(* CODESYS project tc3_hbi_system.library
   Company: BeckHoff
   DefaultNamespace: Tc3_HBI_System
   Version: 3.3.2.1
   Placeholder: Tc3_HBI_System
   Title: Tc3_HBI_System

Project tree, tasks and I/O mapping:
  libraries: Tc2_EtherCAT, * (Beckhoff Automation GmbH); Tc2_IoFunctions, * (Beckhoff Automation GmbH); Tc2_Standard, * (Beckhoff Automation GmbH); Tc2_SUPS, * (Beckhoff Automation GmbH); Tc2_System, * (Beckhoff Automation GmbH); Tc2_Utilities, * (Beckhoff Automation GmbH); Tc3_Interfaces, * (Beckhoff Automation GmbH); Tc3_Module, * (Beckhoff Automation GmbH)
  DUTs/
  GVLs/
  POUs/
    BASIC/
      POUs/
        FBs/
          DUTs/
            data type ST_Basic
            data type ST_Basic_Status
          GVLs/
            global variables GVL_Basic
          ITFs/
            interface I_Basic: M_nError, M_nReset, P_bAuto, P_bError, P_bManual, P_bReady, P_bReset, P_nErrorID
          function block FB_Basic [ST]: M_nError, M_nReset, P_bAuto, P_bError, P_bManual, P_bReady, P_bReset, P_nErrorID
    FileSystem/
      ITFs/
        interface I_FileSystem: P_sDirectoryPath, P_sSubDirPath
      DUTs/
        data type ST_FileSystem
      function block FB_FileAccess [ST]: M_nDirectory, M_nSequence, M_sGetToken, P_sDirectoryPath, P_sSubDirPath
    SYSTEM/
      POUs/
        FBs/
          EtherCAT/
            DUTs/
              HW/
                data type ST_EtherCAT_HW_IN
                data type ST_EtherCAT_HW_TerminalDiagInfo
              data type ST_EtherCAT_Diag
              data type ST_EtherCAT_HW_Diag
            GVLs/
              global variables GVL_EtherCAT_Diag
            ITFs/
              interface I_EtherCAT_Diag: M_nCyclic, P_bEtherCAT_Ok, P_bWcError, P_nCfgSlaveCount, P_nDevState, P_nSlaveCounts
            function block FB_EtherCAT_Diag [ST]: M_nCyclic, M_sGetToken, P_bEtherCAT_Ok, P_bWcError, P_nCfgSlaveCount, P_nDevState, P_nSlaveCounts
          NovRam/
            DUTs/
              data type ST_NovRam
            ITFs/
              interface I_NovRam: M_nEnable
            function block FB_NovRam [ST]: M_nEnable, M_nRead, M_nWrite
          Persistent/
            DUTs/
              data type ST_WritePersistentData
            ITFs/
              interface I_WritePersistentData: M_n1_Second_UPS, M_nEnable, M_nWrite, P_bBusy, P_bPowerFailDetect, P_eSUPS_Mode, P_nWriteCNT
            function block FB_WritePersistentData [ST]: M_n1_Second_UPS, M_nEnable, M_nWrite, P_bBusy, P_bPowerFailDetect, P_eSUPS_Mode, P_nWriteCNT
          System/
            DUTs/
              data type ST_System
            ITFs/
              interface I_System: M_nCerHost, M_nEnable, M_nGetTimeStampInMs, P_bIs_ARM, P_bIs_CE_Device, P_bIs_x64, P_bIs_x86, P_nAdsPort, P_nCycleTime, P_stDeviceIdentificationEx, P_sTwinCAT_Version
            function block FB_System [ST]: M_nCerHost, M_nEnable, M_nGetTimeStampInMs, P_bIs_ARM, P_bIs_CE_Device, P_bIs_x64, P_bIs_x86, P_nAdsPort, P_nCycleTime, P_stDeviceIdentificationEx, P_sTwinCAT_Version
  Version/
    global variables Global_Version
  VISUs/
  Tc3_HBI_System.tmc
*)

// POUs/BASIC/POUs/FBs/DUTs/ST_Basic
TYPE ST_Basic :
STRUCT
	bAuto: BOOL;
	bManual: BOOL;
	bReady: BOOL;
	bReset: BOOL;
	bError: BOOL;
	nErrorID: UDINT;
	nStatus: UDINT;	
	arr_nStatus: ARRAY[1..20] OF UDINT;
END_STRUCT
END_TYPE

// POUs/BASIC/POUs/FBs/DUTs/ST_Basic_Status
TYPE ST_Basic_Status :
STRUCT
	nError: UDINT;
	nReset:UDINT;
END_STRUCT
END_TYPE

// POUs/FileSystem/DUTs/ST_FileSystem
TYPE ST_FileSystem :
STRUCT
END_STRUCT
END_TYPE

// POUs/SYSTEM/POUs/FBs/EtherCAT/DUTs/HW/ST_EtherCAT_HW_IN
TYPE ST_EtherCAT_HW_IN :
STRUCT
	AI_AmsNetId: AMSNETID;
	AI_nDevState: UINT;
	AI_nCfgSlaveCount: UINT;							
	AI_nSlaveCounts: UINT;								
	AI_nFrmXWcState: ARRAY[0..(GVL_EtherCAT_Diag.MAX_NUMBERS_OF_EC_FRAMES -1)] OF UINT;
END_STRUCT
END_TYPE

// POUs/SYSTEM/POUs/FBs/EtherCAT/DUTs/HW/ST_EtherCAT_HW_TerminalDiagInfo
TYPE ST_EtherCAT_HW_TerminalDiagInfo :
STRUCT
	nAddr: UINT;
	sType: STRING(50);
	sName: STRING(50);
	nDeviceState: BYTE;
	nLinkState: BYTE;
END_STRUCT
END_TYPE

// POUs/SYSTEM/POUs/FBs/EtherCAT/DUTs/ST_EtherCAT_Diag
TYPE ST_EtherCAT_Diag EXTENDS ST_Basic:
STRUCT
	bEtherCAT_Ok: BOOL;				// ErtherCAT Ok signal
	bWcError: BOOL;
	nDevState: UINT;
	nCfgSlaveCount: UINT;							
	nSlaveCounts: UINT;								
END_STRUCT
END_TYPE

// POUs/SYSTEM/POUs/FBs/EtherCAT/DUTs/ST_EtherCAT_HW_Diag
TYPE ST_EtherCAT_HW_Diag :
STRUCT
	stAmsNetId: AMSNETID;			// EtherCAT Ams net id
	nState: WORD;					// EtherCAT master state
	sState: STRING;					// EtherCAT master state (string)
	nDevState: UINT;				// EtherCAT master DevState
	sDevState: STRING;				// EtherCAT master DevState (string)
	nCfgSlaveCount: UINT;			// Project configured slaves
	nSlaveCounts: UINT;				// Actual slave counts
	nMaxNumberOfSlaves: UINT;		// Max numbers of EtherCAT slaves
	bWcError: BOOL;					// Wc error
	bEtherCAT_Ok: BOOL;				// ErtherCAT Ok signal
	bReady: BOOL;					// Ready
	bError: BOOL;					// Error
	nErrorID: UDINT;				// Error ID
	arrFrmXWcState: ARRAY[0..(GVL_EtherCAT_Diag.MAX_NUMBERS_OF_EC_FRAMES - 1)] OF UINT;		// EtherCAT master Wc state
	arrEcTerminalDiagInfo: ARRAY[1..GVL_EtherCAT_Diag.MAX_NUMBERS_OF_EC_SLAVES] OF ST_EtherCAT_HW_TerminalDiagInfo;
END_STRUCT
END_TYPE

// POUs/SYSTEM/POUs/FBs/NovRam/DUTs/ST_NovRam
TYPE ST_NovRam EXTENDS ST_Basic :
STRUCT
	bEnable: BOOL;
END_STRUCT
END_TYPE

// POUs/SYSTEM/POUs/FBs/Persistent/DUTs/ST_WritePersistentData
TYPE ST_WritePersistentData EXTENDS ST_Basic :
STRUCT
	bWrite: BOOL;
	bBusy: BOOL;
	bPowerFailDetect: BOOL;
	nWriteCNT: UDINT;
END_STRUCT
END_TYPE

// POUs/SYSTEM/POUs/FBs/System/DUTs/ST_System
TYPE ST_System EXTENDS ST_Basic :
STRUCT
	bIs_CE_Device: BOOL;			// Is a CE Device
	bIs_ARM: BOOL;					// Is ARM runtime
	bIs_x86: BOOL;					// Is x86 runtime
	bIs_x64: BOOL;					// Is x64 runtime
	nAdsPort: UINT;					// Plc port nr
	nCycleTime: UDINT;				// Plc cycle time in 100nS
	bCerHost_Enable: BOOL;			// Enable CerHost
	bCerHost_Disable: BOOL;			// Disable CerHost
	sTwinCAT_Version: STRING(20);	// Runtime version
	stDeviceIdentificationEx: Tc2_Utilities.ST_DeviceIdentificationEx;
END_STRUCT
END_TYPE

// POUs/BASIC/POUs/FBs/GVLs/GVL_Basic
VAR_GLOBAL CONSTANT
	cIDLE: UDINT:= 0;						//	0 = idle
	cCOUPLED: UDINT:= 1;					//	1 = coupled
	cSTARTING: UDINT:= 2;					//	2 = starting
	cRUNNING: UDINT:= 3;					//	3 = running
	cABORTED: UDINT:= 4;					//	4 = aborted
	cNO_HARDWARE_CONNECTED: UDINT:= 5;		// 	5 = no hardware connected

	cPOINTER_OR_INDEX_ERROR: UDINT:= 7;		//	7 = pointer or index error
	cMAPPING_ERROR: UDINT:= 8;				//	8 = mapping error
	cPARAMETER_ERROR: UDINT:= 9;			//	9 = parameter error
	cCOMPLETE: UDINT:= 10;					//	10 = complete
END_VAR

// POUs/SYSTEM/POUs/FBs/EtherCAT/GVLs/GVL_EtherCAT_Diag
{attribute 'qualified_only'}
VAR_GLOBAL CONSTANT
	MAX_NUMBERS_OF_EC_SLAVES: UINT:= 1000;		// Max numbers of EtherCAT slaves
	MAX_NUMBERS_OF_EC_FRAMES: UINT:= 10;		// Max numbers of EtherCAT frames
END_VAR

// Version/Global_Version
{attribute 'TcGenerated'}
// This function has been automatically generated from the project information.
VAR_GLOBAL CONSTANT
	{attribute 'const_non_replaced'}
	{attribute 'linkalways'}
	stLibVersion_Tc3_HBI_System : ST_LibVersion := (iMajor := 3, iMinor := 3, iBuild := 2, iRevision := 1, sVersion := '3.3.2.1');
END_VAR

// POUs/BASIC/POUs/FBs/ITFs/I_Basic
INTERFACE I_Basic

//	The result of the method is an unsigned double integer
//	0 = idle 
//	1 = coupled
//	2 = starting
//	3 = running
//	4 = aborted
// 	5 = no hardware connected
//  6 = Spare
//	7 = pointer or index error
//	8 = mapping error
//	9 = parameter error
//	10 = complete
//	Any other number = ErrorID
METHOD PUBLIC M_nError : UDINT
VAR_INPUT
	nErrorID: UDINT;
END_VAR
END_METHOD

//	The result of the method is an unsigned double integer
//	0 = idle 
//	1 = coupled
//	2 = starting
//	3 = running
//	4 = aborted
// 	5 = no hardware connected
//  6 = Spare
//	7 = pointer or index error
//	8 = mapping error
//	9 = parameter error
//	10 = complete
//	Any other number = ErrorID
METHOD PUBLIC M_nReset : UDINT
VAR_INPUT
	bExecute: BOOL;
END_VAR
END_METHOD

PROPERTY PUBLIC P_bAuto : BOOL
GET
END_GET
SET
END_SET
END_PROPERTY

PROPERTY PUBLIC P_bError : BOOL
GET
END_GET
END_PROPERTY

PROPERTY PUBLIC P_bManual : BOOL
GET
END_GET
SET
END_SET
END_PROPERTY

PROPERTY PUBLIC P_bReady : BOOL
GET
END_GET
SET
END_SET
END_PROPERTY

PROPERTY PUBLIC P_bReset : BOOL
GET
END_GET
END_PROPERTY

PROPERTY PUBLIC P_nErrorID : UDINT
GET
END_GET
END_PROPERTY

END_INTERFACE

// POUs/BASIC/POUs/FBs/FB_Basic
//------------------------------------------------------------------------------------------
//                                                                                        	
//***************************** Beckhoff TwinCAT Examples **********************************
//                                                                                        	
//************************************* WARNING ********************************************
// This program is only an example. If it is used as a control program in any real        	
// application, Beckhoff is not responsible for any malfunction, loss or damage           	
// which could arise by using this program!                                               	
//                                                                                        	
//*************************************  Program Info. *************************************
//                                                                                        	
// PLC program name:       	FB_Basic (FB)               	                           	
// Hardware platform:      	TwinCat v3.1.4022				                          	                                  	
//                                                                                        	
// ======================================================================================== 
//         Version       Date                        Remarks                              	
// ======================================================================================== 
//         3.1           27 feb 2018                 First release of this example        	    	
// ======================================================================================== 
//                                                                                        	
//******************************* Aims OF this PLC PROGRAM *********************************
//                                                                                        	
// Basic FB  						 			                               	
//																	                      	
//                                                                                        	
//----------------------------------------------------------------------------------------- 
FUNCTION_BLOCK FB_Basic IMPLEMENTS I_Basic
VAR
	_iIdx: INT;		// Temporary variabel - Index pointer
	
//*************************
// Property variables
//*************************
	_bReset: BOOL;
	_bAuto: BOOL := TRUE;
	_bManual: BOOL;
	_bError: BOOL;
	_nErrorID: UDINT;
	_bReady: BOOL;
	
//*************************
// Methods variable
//*************************
	FB_Basic_M_nReset_nScanCNT: UINT;
	FB_Basic_M_nReset_fbR_TRIG: Tc2_Standard.R_TRIG;
END_VAR

//	The result of the method is an unsigned double integer
//	0 = idle 
//	1 = coupled
//	2 = starting
//	3 = running
//	4 = aborted
// 	5 = no hardware connected
//  6 = Spare
//	7 = pointer or index error
//	8 = mapping error
//	9 = parameter error
//	10 = complete
//	Any other number = ErrorID
METHOD PUBLIC M_nError : UDINT
VAR_INPUT
	nErrorID: UDINT;
END_VAR
//**********************************
// Update error
//**********************************
IF NOT _bReset THEN
	IF NOT _bError THEN
		_nErrorID:= nErrorID;
		_bError:= TRUE;
	END_IF
END_IF

M_nError:= cCOMPLETE;
END_METHOD

//	The result of the method is an unsigned double integer
//	0 = idle 
//	1 = coupled
//	2 = starting
//	3 = running
//	4 = aborted
// 	5 = no hardware connected
//  6 = Spare
//	7 = pointer or index error
//	8 = mapping error
//	9 = parameter error
//	10 = complete
//	Any other number = ErrorID
METHOD PUBLIC M_nReset : UDINT
VAR_INPUT
	bExecute: BOOL;
END_VAR
//**********************************
// Wait for execute
//**********************************
FB_Basic_M_nReset_fbR_TRIG(CLK:= bExecute);
IF FB_Basic_M_nReset_fbR_TRIG.Q THEN
	FB_Basic_M_nReset_nScanCNT:= 4;	
	_bReset:= TRUE;
ELSE
	// Delay
	IF FB_Basic_M_nReset_nScanCNT = 0 THEN
		IF NOT bExecute THEN
			_bReset:= FALSE;
		END_IF
	ELSE
		IF FB_Basic_M_nReset_nScanCNT <= 2 THEN
			_bError:= FALSE;
			_nErrorID:= 16#00;
		END_IF	
	END_IF

	// Scan counter
	IF FB_Basic_M_nReset_nScanCNT > 0 THEN
		FB_Basic_M_nReset_nScanCNT:= FB_Basic_M_nReset_nScanCNT -1;
	ELSE	
		FB_Basic_M_nReset_nScanCNT:= 0;
	END_IF

	// Return method state
	IF bExecute THEN
		IF FB_Basic_M_nReset_nScanCNT = 0 THEN
			M_nReset:= cCOMPLETE;
		ELSE
			M_nReset:= cRUNNING;
		END_IF
	ELSE	
		M_nReset:= cIDLE;
	END_IF	
END_IF
END_METHOD

PROPERTY PUBLIC P_bAuto : BOOL
GET
P_bAuto:= _bAuto;
END_GET
SET
_bAuto:= P_bAuto;
END_SET
END_PROPERTY

PROPERTY PUBLIC P_bError : BOOL
GET
P_bError:= _bError;
END_GET
END_PROPERTY

PROPERTY PUBLIC P_bManual : BOOL
GET
P_bManual:= _bManual;
END_GET
SET
_bManual:= P_bManual;
END_SET
END_PROPERTY

PROPERTY PUBLIC P_bReady : BOOL
GET
P_bReady:= _bReady;
END_GET
SET
PUBLIC 
VAR
END_VAR
_bReady:= P_bReady;
END_SET
END_PROPERTY

PROPERTY PUBLIC P_bReset : BOOL
GET
P_bReset:= _bReset;
END_GET
END_PROPERTY

PROPERTY PUBLIC P_nErrorID : UDINT
GET
P_nErrorID:= _nErrorID;
END_GET
END_PROPERTY

END_FUNCTION_BLOCK

// POUs/FileSystem/ITFs/I_FileSystem
INTERFACE I_FileSystem EXTENDS I_Basic

PROPERTY P_sDirectoryPath : T_MaxString
GET
END_GET
SET
END_SET
END_PROPERTY

PROPERTY P_sSubDirPath : T_MaxString
GET
END_GET
SET
END_SET
END_PROPERTY

END_INTERFACE

// POUs/FileSystem/FB_FileAccess
FUNCTION_BLOCK PUBLIC FB_FileAccess EXTENDS FB_Basic IMPLEMENTS I_FileSystem
VAR_INPUT
END_VAR
VAR_OUTPUT
END_VAR
VAR
	// Directory
	FB_FileAccess_DirectoryPath:	T_MAXSTRING:='C:\';
	FB_FileAccess_SubDirPath:		T_MAXSTRING:='AEM\Data\ControllerLog';
	fbCreateDir			: FB_CreateDir;
	fbEnumFindFileEntry	: FB_EnumFindFileEntry;
	
	FB_FileAccess_M_nDirectory_iState	: INT;
	FB_FileAccess_M_nDirectory_bExecute: BOOL;
	FB_FileAccess_M_nDirectory_fbExecute: R_TRIG;
	
	FB_FileAccess_M_nSequence_iState	: INT;
	FB_FileAccess_M_nSequence_bExecute: BOOL;
	FB_FileAccess_M_nSequence_fbExecute: R_TRIG;
	FB_FileAccess_M_nSequence_sPathName:	T_MAXSTRING:='C:\AEM\Data\ControllerLog';
	
	FB_FileAccess_M_nDirectory_sSubDirPath: T_MAXSTRING;
	FB_FileAccess_M_nDirectory_sSubDirPath1: T_MAXSTRING;
	FB_FileAccess_M_nDirectory_sSubDirPath2: T_MAXSTRING;
	FB_FileAccess_M_nDirectory_sSubDirPath3: T_MAXSTRING;
	FB_FileAccess_M_nDirectory_sSubDirPath4: T_MAXSTRING;
	FB_FileAccess_M_nDirectory_nToken	   : INT;	
END_VAR

METHOD PUBLIC M_nDirectory : UDINT
VAR_INPUT
	bExecute: BOOL;
END_VAR
VAR	
END_VAR
FB_FileAccess_M_nDirectory_bExecute:= bExecute;
FB_FileAccess_M_nDirectory_fbExecute(CLK:= FB_FileAccess_M_nDirectory_bExecute, Q=> );

IF FB_FileAccess_M_nDirectory_fbExecute.Q THEN
	FB_FileAccess_M_nDirectory_iState:= 10;
END_IF

	FB_FileAccess_M_nDirectory_sSubDirPath1:= M_sGetToken(sAllTokens:= FB_FileAccess_SubDirPath, nToken:= 1, sDelim:= '\');
	FB_FileAccess_M_nDirectory_sSubDirPath2:= M_sGetToken(sAllTokens:= FB_FileAccess_SubDirPath, nToken:= 2, sDelim:= '\');
	FB_FileAccess_M_nDirectory_sSubDirPath3:= M_sGetToken(sAllTokens:= FB_FileAccess_SubDirPath, nToken:= 3, sDelim:= '\');
	FB_FileAccess_M_nDirectory_sSubDirPath4:= M_sGetToken(sAllTokens:= FB_FileAccess_SubDirPath, nToken:= 4, sDelim:= '\');
	
	IF FB_FileAccess_M_nDirectory_sSubDirPath1='' OR FB_FileAccess_M_nDirectory_sSubDirPath2= '' OR FB_FileAccess_M_nDirectory_sSubDirPath3=''
			OR FB_FileAccess_M_nDirectory_sSubDirPath4<> '' THEN
		M_nError(nErrorID:= cPARAMETER_ERROR);
		M_nDirectory:= cPARAMETER_ERROR;
		RETURN;
	END_IF
	
IF _bReset THEN
	IF _bError THEN
		FB_FileAccess_M_nDirectory_iState:= 0;
	END_IF
END_IF

CASE FB_FileAccess_M_nDirectory_iState OF
 
	0: // Init
		M_nDirectory:= cIDLE;
		
		M_nSequence(bExecute:= FALSE, sPathName:= 'C:\AEM\Data\ControllerLog');
		FB_FileAccess_M_nDirectory_iState:= 1;
		
	1: // Waiting for execute
		;
		
	10: // Create directory
	
		M_nDirectory:= cRUNNING;
		
		IF M_nSequence(bExecute:= TRUE, sPathName:= CONCAT(FB_FileAccess_DirectoryPath,FB_FileAccess_M_nDirectory_sSubDirPath1))= cComplete THEN
			M_nSequence(bExecute:= FALSE, sPathName:= CONCAT(FB_FileAccess_DirectoryPath,FB_FileAccess_M_nDirectory_sSubDirPath1));
			FB_FileAccess_M_nDirectory_iState:= 20;
			ELSIF _bError THEN
				M_nDirectory:= M_nError(nErrorID:= _nErrorID);
				FB_FileAccess_M_nDirectory_iState:= 999;
		END_IF
	
	20: // Create directory
		M_nDirectory:= cRUNNING;
		IF M_nSequence(bExecute:= TRUE, sPathName:= CONCAT(FB_FileAccess_DirectoryPath,
				CONCAT(FB_FileAccess_M_nDirectory_sSubDirPath1,CONCAT('\',FB_FileAccess_M_nDirectory_sSubDirPath2))))= cComplete THEN
			M_nSequence(bExecute:= FALSE, sPathName:= CONCAT(FB_FileAccess_DirectoryPath,FB_FileAccess_M_nDirectory_sSubDirPath1));
			FB_FileAccess_M_nDirectory_iState:= 30;
			ELSIF _bError THEN
				M_nDirectory:= M_nError(nErrorID:= _nErrorID);
				FB_FileAccess_M_nDirectory_iState:= 999;
		END_IF
	
	30: // Create directory
		M_nDirectory:= cRUNNING;
		IF M_nSequence(bExecute:= TRUE, sPathName:= CONCAT(FB_FileAccess_DirectoryPath,CONCAT(FB_FileAccess_M_nDirectory_sSubDirPath1,
							CONCAT('\',CONCAT(FB_FileAccess_M_nDirectory_sSubDirPath2,CONCAT('\',FB_FileAccess_M_nDirectory_sSubDirPath3))))))= cComplete THEN
			M_nSequence(bExecute:= FALSE, sPathName:= CONCAT(FB_FileAccess_DirectoryPath,FB_FileAccess_M_nDirectory_sSubDirPath1));
			FB_FileAccess_M_nDirectory_iState:= 40;
			ELSIF _bError THEN
				M_nDirectory:= M_nError(nErrorID:= _nErrorID);
				FB_FileAccess_M_nDirectory_iState:= 999;
		END_IF
		
	40:
		M_nDirectory:= cComplete;
		
		IF NOT FB_FileAccess_M_nDirectory_bExecute THEN
			FB_FileAccess_M_nDirectory_iState:= 0;
		END_IF
	
	999:// Error state
		M_nSequence(bExecute:= FALSE, sPathName:= CONCAT(FB_FileAccess_DirectoryPath,FB_FileAccess_M_nDirectory_sSubDirPath1));
		
	ELSE FB_FileAccess_M_nDirectory_iState:= 0;
		
END_CASE
END_METHOD

METHOD PUBLIC M_nSequence : UDINT
VAR_INPUT
	bExecute: BOOL;
	sPathName: T_MaxString;
END_VAR
// Local variables
FB_FileAccess_M_nSequence_bExecute:= bExecute;
FB_FileAccess_M_nSequence_sPathName:= sPathName;

IF _bReset THEN
	IF _bError THEN
		FB_FileAccess_M_nSequence_iState:= 0;
	END_IF
END_IF

FB_FileAccess_M_nSequence_fbExecute(CLK:= FB_FileAccess_M_nSequence_bExecute, Q=> );
IF FB_FileAccess_M_nSequence_fbExecute.Q THEN
	FB_FileAccess_M_nSequence_iState:= 10;
END_IF

CASE FB_FileAccess_M_nSequence_iState OF 
	0: // Init
		M_nSequence:= cIDLE;
		
		fbEnumFindFileEntry(sNetId:= '', bExecute:= FALSE, );
		fbCreateDir(sNetId:= '', bExecute:= FALSE, );
		FB_FileAccess_M_nSequence_iState:= 1;
		
	1: // Waiting for execute
		;
		
	10: // Check if directory exit
		M_nSequence:= cRUNNING;
		
		fbEnumFindFileEntry(
			sNetId:= '', 
			sPathName:= FB_FileAccess_M_nSequence_sPathName, 
			eCmd:= eEnumCmd_First, 
			bExecute:= TRUE, 
			tTimeout:= T#5S, 
			bBusy=> , 
			bError=> , 
			nErrID=> , 
			bEOE=> , 
			stFindFile=> );
		IF NOT fbEnumFindFileEntry.bBusy THEN	
			IF fbEnumFindFileEntry.bError THEN
				M_nError(nErrorID:= fbEnumFindFileEntry.nErrId);
				FB_FileAccess_M_nSequence_iState:= 999;
			ELSE
				IF NOT fbEnumFindFileEntry.bEOE THEN
					FB_FileAccess_M_nSequence_iState:= 30; (*target dir is exist*)
					ELSE 
						FB_FileAccess_M_nDirectory_sSubDirPath:= FB_FileAccess_M_nSequence_sPathName;
						FB_FileAccess_M_nSequence_iState:= 20;	(*target dir no exist*)
				END_IF
			END_IF
			fbEnumFindFileEntry(sNetId:= '', bExecute:= FALSE, );
		END_IF	
		
	20: // Create directory
		M_nSequence:= cRUNNING;
		
		fbCreateDir(
			sNetId:= '', 
			sPathName:= FB_FileAccess_M_nSequence_sPathName, 
			ePath:= PATH_GENERIC, 
			bExecute:= TRUE, 
			tTimeout:= T#5S, 
			bBusy=> , 
			bError=> , 
			nErrId=> );
		IF NOT fbCreateDir.bBusy THEN	
			IF fbCreateDir.bError THEN
				M_nError(nErrorID:= fbCreateDir.nErrId);
				FB_FileAccess_M_nSequence_iState:= 999;
			ELSE
				FB_FileAccess_M_nSequence_iState:= 30;	
			END_IF
			fbCreateDir(sNetId:= '', bExecute:= FALSE, );
		END_IF
		
	30: // Complete
		M_nSequence:= cComplete;
		IF NOT FB_FileAccess_M_nSequence_bExecute THEN
			FB_FileAccess_M_nSequence_iState:= 0;
		END_IF
		
	999: // error state
		;
	
	ELSE FB_FileAccess_M_nSequence_iState:= 0;
		
END_CASE
END_METHOD

METHOD PUBLIC M_sGetToken : STRING
VAR_INPUT
	sAllTokens: Tc2_System.T_MaxString;
	nToken: UINT;
  	sDelim: STRING;
END_VAR
VAR
// Temporary Variables 
	pString: POINTER TO STRING;
	nCurTokenLocation: INT;
END_VAR
pString:= ADR(sAllTokens);

IF nToken < 1 OR LEN(sDelim) < 1 THEN
	// Negative OR zeroth token OR empty delimiter strings mean an empty token 
	M_sGetToken:= '';
 	RETURN;
ELSE
	IF nToken = 1 THEN
	// Quickly extract the first token 
	nCurTokenLocation:= FIND(pString^, sDelim);
	   	IF nCurTokenLocation > 1 THEN
	   		M_sGetToken:= LEFT(pString^, nCurTokenLocation - 1);
	   	ELSE
			M_sGetToken:= pString^;
	    END_IF
	ELSE
		// FIND the Nth token 
		REPEAT
			nCurTokenLocation:= FIND(pString^, sDelim);
			IF nCurTokenLocation = 0 THEN
				M_sGetToken:= '';
				RETURN;
			ELSE
				pString:= pString + INT_TO_DWORD(nCurTokenLocation -1) + INT_TO_DWORD(LEN(sDelim));
			END_IF
	
			nToken:= nToken - 1;
			UNTIL nToken = 1
		END_REPEAT;

		// Extract the Nth token (Which is the next token AT this point) 
		nCurTokenLocation:= FIND(pString^, sDelim);
		IF nCurTokenLocation > 0 THEN
			M_sGetToken:= LEFT(pString^, nCurTokenLocation - 1);
			RETURN;
		ELSE
			M_sGetToken:= pString^;
		   	RETURN;
		END_IF
	END_IF
END_IF
END_METHOD

PROPERTY P_sDirectoryPath : T_MaxString
GET
P_sDirectoryPath:= FB_FileAccess_DirectoryPath;
END_GET
SET
FB_FileAccess_DirectoryPath:= P_sDirectoryPath;
END_SET
END_PROPERTY

PROPERTY P_sSubDirPath : T_MaxString
GET
P_sSubDirPath:= FB_FileAccess_SubDirPath;
END_GET
SET
FB_FileAccess_SubDirPath:= P_sSubDirPath;
END_SET
END_PROPERTY

END_FUNCTION_BLOCK

// POUs/SYSTEM/POUs/FBs/EtherCAT/ITFs/I_EtherCAT_Diag
INTERFACE I_EtherCAT_Diag EXTENDS I_Basic

//	The result of the method is an unsigned double integer
//	0 = idle 
//	1 = coupled
//	2 = starting
//	3 = running
//	4 = aborted
// 	5 = no hardware connected
//  6 = Spare
//	7 = pointer or index error
//	8 = mapping error
//	9 = parameter error
//	10 = complete
//	Any other number = ErrorID
METHOD PUBLIC M_nCyclic : UDINT
VAR_INPUT
	bEnable: BOOL;
	pEtherCAT_Diag: POINTER TO ST_EtherCAT_HW_Diag;	
END_VAR
END_METHOD

PROPERTY PUBLIC P_bEtherCAT_Ok : BOOL
GET
END_GET
SET
END_SET
END_PROPERTY

PROPERTY PUBLIC P_bWcError : bool
GET
END_GET
END_PROPERTY

PROPERTY PUBLIC P_nCfgSlaveCount : UINT
GET
END_GET
END_PROPERTY

PROPERTY PUBLIC P_nDevState : UINT
GET
END_GET
END_PROPERTY

PROPERTY PUBLIC P_nSlaveCounts : UINT
GET
END_GET
END_PROPERTY

END_INTERFACE

// POUs/SYSTEM/POUs/FBs/EtherCAT/FB_EtherCAT_Diag
//------------------------------------------------------------------------------------------
//                                                                                        	
//***************************** Beckhoff TwinCAT Examples **********************************
//                                                                                        	
//************************************* WARNING ********************************************
// This program is only an example. If it is used as a control program in any real        	
// application, Beckhoff is not responsible for any malfunction, loss or damage           	
// which could arise by using this program!                                               	
//                                                                                        	
//*************************************  Program Info. *************************************
//                                                                                        	
// PLC program name:       	FB_EtherCAT_Diag (FB)                                          	
// Hardware platform:      	TwinCAT v3.1.4022				                          	                                  	
//                                                                                        	
// ======================================================================================== 
//         Version       Date                        Remarks                              	
// ======================================================================================== 
//         3.1           27 feb 2018                 First release of this example        	
// ======================================================================================== 
//                                                                                        	
//******************************* Aims OF this PLC PROGRAM *********************************
//                                                                                        	
// EtherCAT diagnose				 			                                      	
//																	                      	
//                                                                                        	
//----------------------------------------------------------------------------------------- 
FUNCTION_BLOCK FB_EtherCAT_Diag EXTENDS FB_Basic IMPLEMENTS I_EtherCAT_Diag
VAR
	bFirstScan: BOOL:= TRUE;
	stIN AT %I*: ST_EtherCAT_HW_IN;
	
	_pEtherCAT_Diag: POINTER TO ST_EtherCAT_HW_Diag;	
	_bWcError: BOOL;
	_nDeviceNumber: UINT:= 1;
	
	arrEcSlaveConfigData: ARRAY[1..GVL_EtherCAT_Diag.MAX_NUMBERS_OF_EC_SLAVES] OF Tc2_EtherCAT.ST_EcSlaveConfigData;
	arrEcSlaveState: ARRAY[1..GVL_EtherCAT_Diag.MAX_NUMBERS_OF_EC_SLAVES] OF Tc2_EtherCAT.ST_EcSlaveState;
	arrEcSlaveName: ARRAY[1..GVL_EtherCAT_Diag.MAX_NUMBERS_OF_EC_SLAVES] OF STRING;;

	fbEcGetMasterState: Tc2_EtherCAT.FB_EcGetMasterState;
	fbEcGetConfSlaves: Tc2_EtherCAT.FB_EcGetConfSlaves;
	fbEcGetAllSlaveStates: Tc2_EtherCAT.FB_EcGetAllSlaveStates;
	fbEcGetSlaveIdentity: Tc2_EtherCAT.FB_EcGetSlaveIdentity;
END_VAR

//	The result of the method is an unsigned double integer
//	0 = idle 
//	1 = coupled
//	2 = starting
//	3 = running
//	4 = aborted
// 	5 = no hardware connected
//  6 = Spare
//	7 = pointer or index error
//	8 = mapping error
//	9 = parameter error
//	10 = complete
//	Any other number = ErrorID
METHOD PUBLIC M_nCyclic : UDINT
VAR_INPUT
	bEnable: BOOL;
	pEtherCAT_Diag: POINTER TO ST_EtherCAT_HW_Diag;	
END_VAR
VAR_INST
	i: UINT;
	iState: INT;
	sString: STRING;
	nDevStateOld: UINT;
	nSlaveCountsOld: UINT;								
	arrFrmXWcStateOld: ARRAY[0..(GVL_EtherCAT_Diag.MAX_NUMBERS_OF_EC_FRAMES -1)] OF UINT;
	arrFrmXWcStateInit: ARRAY[0..(GVL_EtherCAT_Diag.MAX_NUMBERS_OF_EC_FRAMES -1)] OF UINT;
	fbEnable_R_TRIG: Tc2_Standard.R_TRIG;
END_VAR
// Local variable
_pEtherCAT_Diag:= pEtherCAT_Diag;

// Reset
IF _bReset THEN
	IF NOT P_bReady THEN
		iState:= 000;
	END_IF	
END_IF

// Pointer check
IF _pEtherCAT_Diag = 16#00 THEN
	_bReady:= FALSE;
	iState:= 000;
	M_nCyclic:= cPOINTER_OR_INDEX_ERROR;
	RETURN;
END_IF

// EtherCAT Mapping check
IF stIN.AI_AmsNetId[0] = 0 AND stIN.AI_AmsNetId[5] = 0 THEN
	_bReady:= FALSE;
	iState:= 000;
	M_nCyclic:= cMAPPING_ERROR;
	RETURN;
END_IF

// Mapping check
IF stIN.AI_nSlaveCounts = 0 OR stIN.AI_nCfgSlaveCount = 0 THEN
	_bReady:= FALSE;
	iState:= 000;
	M_nCyclic:= cMAPPING_ERROR;
	RETURN;
END_IF

// Not Enable
fbEnable_R_TRIG(CLK:= NOT bEnable, Q=> );
IF fbEnable_R_TRIG.Q THEN
	_bReady:= FALSE;
	iState:= 000;
	RETURN;
END_IF

// Update GVL data
pEtherCAT_Diag^.stAmsNetId:= stIN.AI_AmsNetId;
pEtherCAT_Diag^.bReady:= P_bReady;
pEtherCAT_Diag^.bError:= P_bError;
pEtherCAT_Diag^.nErrorID:= P_nErrorID;
pEtherCAT_Diag^.nMaxNumberOfSlaves:= GVL_EtherCAT_Diag.MAX_NUMBERS_OF_EC_SLAVES;


// State maschine
CASE iState OF
	
	000:	// Init
			fbEcGetMasterState(bExecute:= FALSE); 
			fbEcGetConfSlaves(pArrEcConfSlaveInfo:= ADR(arrEcSlaveConfigData), cbBufLen:= SIZEOF(arrEcSlaveConfigData), bExecute:= FALSE); 
			fbEcGetAllSlaveStates(pStateBuf:= ADR(arrEcSlaveState), cbBufLen:= SIZEOF(arrEcSlaveState), bExecute:= FALSE); 
			fbEcGetSlaveIdentity(bExecute:= FALSE); 
			MEMCPY(destAddr:= ADR(arrFrmXWcStateOld), srcAddr:= ADR(pEtherCAT_Diag^.arrFrmXWcState), n:= SIZEOF(arrFrmXWcStateOld));
			nDevStateOld:= stIN.AI_nDevState;
			nSlaveCountsOld:= stIN.AI_nSlaveCounts;
			P_bReady:= FALSE;
			iState:= iState +1;	

	001:	// Wait for enable	
			IF bEnable THEN
				IF bFirstScan THEN
					iState:= iState +1;
				ELSE
					iState:= iState +2;
				END_IF	
			END_IF
		
	002:	// Get Conf Slaves
			M_nCyclic:= cRUNNING;
			fbEcGetConfSlaves(
				sNetId:= F_CreateAmsNetId(stIN.AI_AmsNetId), 
				pArrEcConfSlaveInfo:= ADR(arrEcSlaveConfigData), 
				cbBufLen:= SIZEOF(arrEcSlaveConfigData), 
				bExecute:= TRUE, 
				tTimeout:= , 
				bBusy=> , 
				bError=> , 
				nErrorId=> , 
				nSlaves=> );
				
			// Error	
			IF fbEcGetConfSlaves.bError THEN
				M_nError(nErrorID:= fbEcGetConfSlaves.nErrorId);
				M_nCyclic:= fbEcGetConfSlaves.nErrorId;
			ELSE
				// Done
				IF NOT fbEcGetConfSlaves.bBusy THEN
					fbEcGetConfSlaves(pArrEcConfSlaveInfo:= ADR(arrEcSlaveConfigData), cbBufLen:= SIZEOF(arrEcSlaveConfigData), bExecute:= FALSE);
					iState:= iState +1;	
				END_IF
			END_IF

	003:	// Get Master state
			M_nCyclic:= cRUNNING;
			fbEcGetMasterState(
				sNetId:= F_CreateAmsNetId(stIN.AI_AmsNetId), 
				bExecute:= TRUE, 
				tTimeout:= , 
				bBusy=> , 
				bError=> , 
				nErrId=> , 
				state=> );

			// Error
			IF fbEcGetMasterState.bError THEN
				M_nError(nErrorID:= fbEcGetMasterState.nErrId);
				M_nCyclic:= fbEcGetMasterState.nErrId;
			ELSE
				// Done
				IF NOT fbEcGetMasterState.bBusy THEN
					fbEcGetMasterState(bExecute:= FALSE); 
					iState:= iState +1;	
				END_IF
			END_IF

	004:	// Get all slave states
			M_nCyclic:= cRUNNING;
			fbEcGetAllSlaveStates(
				sNetId:= F_CreateAmsNetId(stIN.AI_AmsNetId),
				pStateBuf:= ADR(arrEcSlaveState), 
				cbBufLen:= SIZEOF(arrEcSlaveState), 
				bExecute:= TRUE, 
				tTimeout:= , 
				bBusy=> , 
				bError=> , 
				nErrId=> , 
				nSlaves=>);
	
			// Error
			IF fbEcGetAllSlaveStates.bError THEN
				M_nError(nErrorID:= fbEcGetAllSlaveStates.nErrId);
				M_nCyclic:= fbEcGetAllSlaveStates.nErrId;
			ELSE
				// Done	
				IF NOT fbEcGetAllSlaveStates.bBusy THEN
					fbEcGetAllSlaveStates(pStateBuf:= ADR(arrEcSlaveState), cbBufLen:= SIZEOF(arrEcSlaveState), bExecute:= FALSE);
					iState:= iState +1;	
				END_IF 
			END_IF		
				
	005:	// Get device name	
			IF _nDeviceNumber <= fbEcGetAllSlaveStates.nSlaves THEN
				fbEcGetSlaveIdentity(
					sNetId:= F_CreateAmsNetId(stIN.AI_AmsNetId), 
					nSlaveAddr:= arrEcSlaveConfigData[_nDeviceNumber].nAddr, 
					bExecute:= TRUE, 
					tTimeout:= , 
					bBusy=> , 
					bError=> , 
					nErrId=> , 
					identity=> );
		
					// Error
					IF fbEcGetSlaveIdentity.bError THEN
						M_nError(nErrorID:= fbEcGetSlaveIdentity.nErrId);
						M_nCyclic:= fbEcGetSlaveIdentity.nErrId;
					ELSE
						// Done	
						IF NOT fbEcGetSlaveIdentity.bBusy THEN
							arrEcSlaveName[_nDeviceNumber]:= F_ConvProductCodeToString(fbEcGetSlaveIdentity.identity);	
							fbEcGetSlaveIdentity(bExecute:= FALSE); 
							_nDeviceNumber:= _nDeviceNumber +1;
							iState:= iState +1;	
						END_IF 
					END_IF		
				
			ELSE
				iState:= iState +2;	
			END_IF

	006:	// Next device
			iState:= iState -1;	
	
	007:	// Update status
			M_nCyclic:= cRUNNING;

			// Master
			pEtherCAT_Diag^.nState:= fbEcGetMasterState.state;	
			pEtherCAT_Diag^.sState := F_ConvStateToString(fbEcGetMasterState.state);
			pEtherCAT_Diag^.nDevState:= stIN.AI_nDevState; 
			pEtherCAT_Diag^.sDevState:= F_ConvMasterDevStateToString(stIN.AI_nDevState);
			pEtherCAT_Diag^.nSlaveCounts:= stIN.AI_nSlaveCounts;
			pEtherCAT_Diag^.nCfgSlaveCount:= stIN.AI_nCfgSlaveCount;
			
			// Slave counts Wc state update
			FOR i:= 1 TO GVL_EtherCAT_Diag.MAX_NUMBERS_OF_EC_FRAMES DO
				pEtherCAT_Diag^.arrFrmXWcState[i]:= stIN.AI_nFrmXWcState[i];
			END_FOR
			
			// Slave counts status update
			FOR i:= 1 TO fbEcGetAllSlaveStates.nSlaves DO
				pEtherCAT_Diag^.arrEcTerminalDiagInfo[i].nAddr:= arrEcSlaveConfigData[i].nAddr;
				pEtherCAT_Diag^.arrEcTerminalDiagInfo[i].sType:= arrEcSlaveName[i];
				
				// Read string until '('
				sString:= M_sGetToken(pSrcAddr:= ADR(arrEcSlaveConfigData[i].sName), sDelim:= '(', nToken:= 1); 
				IF sString = '' THEN
					pEtherCAT_Diag^.arrEcTerminalDiagInfo[i].sName:= arrEcSlaveConfigData[i].sName;
				ELSE
					sString:= Tc2_Standard.CONCAT(sString,'(');
					sString:= Tc2_Standard.CONCAT(sString,Tc2_Standard.MID(_pEtherCAT_Diag^.arrEcTerminalDiagInfo[i].sType, 6, 1));
					sString:= Tc2_Standard.CONCAT(sString,')');
					pEtherCAT_Diag^.arrEcTerminalDiagInfo[i].sName:= sString;
				END_IF
				pEtherCAT_Diag^.arrEcTerminalDiagInfo[i].nDeviceState:= arrEcSlaveState[i].deviceState;
				pEtherCAT_Diag^.arrEcTerminalDiagInfo[i].nLinkState:= arrEcSlaveState[i].linkState;
				
			END_FOR
			bFirstScan:= FALSE; 
			iState:= iState +1;	
			
	008:	// Wait for DevState change	
			IF nDevStateOld <> stIN.AI_nDevState THEN
				iState:= 000;
			ELSE
				// Wait for Slave counts change
				IF nSlaveCountsOld <> stIN.AI_nSlaveCounts THEN
					iState:= 000;
				ELSE
					// Wait for Wc state change			
					IF MEMCMP(pBuf1:= ADR(arrFrmXWcStateOld), pBuf2:= ADR(pEtherCAT_Diag^.arrFrmXWcState), n:= SIZEOF(arrFrmXWcStateOld)) <> 0 THEN
						iState:= 000;
					END_IF
				END_IF	
			END_IF
			IF P_bError THEN
				P_bReady:= FALSE;
				M_nCyclic:= P_nErrorID;
			ELSE
				P_bReady:= TRUE;
				M_nCyclic:= cCOMPLETE;
			END_IF

ELSE
	iState:= 000;
END_CASE

// Update Wc error
IF MEMCMP(pBuf1:= ADR(_pEtherCAT_Diag^.arrFrmXWcState), pBuf2:= ADR(arrFrmXWcStateInit), n:= SIZEOF(_pEtherCAT_Diag^.arrFrmXWcState)) = 0 THEN
	_pEtherCAT_Diag^.bWcError:= FALSE;
	_bWcError:= FALSE;
ELSE
	_pEtherCAT_Diag^.bWcError:= TRUE;
	_bWcError:= TRUE;
END_IF
END_METHOD

//------------------------------------------------------------------------------------------
//                                                                                        	
//***************************** Beckhoff TwinCAT Examples **********************************
//                                                                                        	
//************************************* WARNING ********************************************
// This program is only an example. If it is used as a control program in any real        	
// application, Beckhoff is not responsible for any malfunction, loss or damage           	
// which could arise by using this program!                                               	
//                                                                                        	
//*************************************  Program Info. *************************************
//                                                                                        	
// PLC program name:       F_sGetToken (FUN)               	                           	
// Hardware platform:      TwinCAT v3.1.4022				                          				                                  	
//                                                                                        	
// ======================================================================================== 
//         Version       Date                        Remarks                              	
// ======================================================================================== 
//         3.1          27 feb 2018                 First release of this example        	
// ======================================================================================== 
//                                                                                        	
//******************************* Aims OF this PLC PROGRAM *********************************
//                                                                                        	
// 	Description:																
//																				
//----------------------------------------------------------------------------------------- 
METHOD PRIVATE M_sGetToken: Tc2_System.T_MaxString
VAR_INPUT
	pSrcAddr: POINTER TO Tc2_System.T_MaxString;
  	sDelim: STRING;
	nToken: UINT;
END_VAR
VAR
// Temporary Variables 
	nCurTokenLocation: INT;
END_VAR
IF nToken < 1 OR Tc2_Standard.LEN(sDelim) < 1 THEN
	// Negative OR zeroth token OR empty delimiter strings mean an empty token 
	M_sGetToken:= '';
 	RETURN;
ELSE
	IF nToken = 1 THEN
	// Quickly extract the first token 
	nCurTokenLocation:= Tc2_Standard.FIND(pSrcAddr^, sDelim);
	   	IF nCurTokenLocation > 1 THEN
	   		M_sGetToken:= Tc2_Standard.LEFT(pSrcAddr^, nCurTokenLocation - 1);
	   	ELSE
			M_sGetToken:= pSrcAddr^;
	    END_IF
	ELSE
		// FIND the Nth token 
		REPEAT
			nCurTokenLocation:= Tc2_Standard.FIND(pSrcAddr^, sDelim);
			IF nCurTokenLocation = 0 THEN
				M_sGetToken:= '';
				RETURN;
			ELSE
				pSrcAddr:= pSrcAddr + INT_TO_DWORD(nCurTokenLocation -1) + INT_TO_DWORD(Tc2_Standard.LEN(sDelim));
			END_IF
	
			nToken:= nToken - 1;
			UNTIL nToken = 1
		END_REPEAT;

		// Extract the Nth token (Which is the next token AT this point) 
		nCurTokenLocation:= Tc2_Standard.FIND(pSrcAddr^, sDelim);
		IF nCurTokenLocation > 0 THEN
			M_sGetToken:= Tc2_Standard.LEFT(pSrcAddr^, nCurTokenLocation - 1);
			RETURN;
		ELSE
			M_sGetToken:= pSrcAddr^;
		   	RETURN;
		END_IF
	END_IF
END_IF
END_METHOD

PROPERTY PUBLIC P_bEtherCAT_Ok : BOOL
GET
// Pointer check
IF _pEtherCAT_Diag <> 16#00 THEN
	P_bEtherCAT_Ok:= _pEtherCAT_Diag^.bEtherCAT_Ok;
ELSE
	P_bEtherCAT_Ok:= FALSE;
END_IF
END_GET
SET
PUBLIC 
VAR
END_VAR
// Pointer check
IF _pEtherCAT_Diag <> 16#00 THEN
	_pEtherCAT_Diag^.bEtherCAT_Ok:= P_bEtherCAT_Ok;
END_IF
END_SET
END_PROPERTY

PROPERTY PUBLIC P_bWcError : bool
GET
P_bWcError:= _bWcError;
END_GET
END_PROPERTY

PROPERTY PUBLIC P_nCfgSlaveCount : UINT
GET
// Pointer check
IF _pEtherCAT_Diag <> 16#00 THEN
	P_nCfgSlaveCount:= _pEtherCAT_Diag^.nCfgSlaveCount;
END_IF
END_GET
END_PROPERTY

PROPERTY PUBLIC P_nDevState : UINT
GET
// Pointer check
IF _pEtherCAT_Diag <> 16#00 THEN
	P_nDevState:= _pEtherCAT_Diag^.nDevState;
END_IF
END_GET
END_PROPERTY

PROPERTY PUBLIC P_nSlaveCounts : UINT
GET
// Pointer check
IF _pEtherCAT_Diag <> 16#00 THEN
	P_nSlaveCounts:= _pEtherCAT_Diag^.nSlaveCounts;
END_IF
END_GET
END_PROPERTY

END_FUNCTION_BLOCK

// POUs/SYSTEM/POUs/FBs/NovRam/ITFs/I_NovRam
INTERFACE I_NovRam EXTENDS I_Basic

//	The result of the method is an unsigned double integer
//	0 = idle 
//	1 = coupled
//	2 = starting
//	3 = running
//	4 = aborted
// 	5 = no hardware connected
//  6 = Spare
//	7 = pointer or index error
//	8 = mapping error
//	9 = parameter error
//	10 = complete
//	Any other number = ErrorID
METHOD M_nEnable : UDINT
VAR_INPUT
	bExecute: BOOL;
	nDevId: UINT;
	nMB_Offset: UINT;
	nMB_Size: UINT;
END_VAR
END_METHOD

END_INTERFACE

// POUs/SYSTEM/POUs/FBs/NovRam/FB_NovRam
//------------------------------------------------------------------------------------------
//                                                                                        	
//***************************** Beckhoff TwinCAT Examples **********************************
//                                                                                        	
//************************************* WARNING ********************************************
// This program is only an example. If it is used as a control program in any real        	
// application, Beckhoff is not responsible for any malfunction, loss or damage           	
// which could arise by using this program!                                               	
//                                                                                        	
//*************************************  Program Info. *************************************
//                                                                                        	
// PLC program name:       	FB_NovRam (FB)               	                           	
// Hardware platform:      	TwinCat v3.1.4022				                          	                                  	
//                                                                                        	
// ======================================================================================== 
//         Version       Date                        Remarks                              	
// ======================================================================================== 
//         3.1           27 feb 2018                 First release of this example        	
// ======================================================================================== 
//                                                                                        	
//******************************* Aims OF this PLC PROGRAM *********************************
//                                                                                        	
//	Read/Write to NovRam																	                      	
//                                                                                        	
//----------------------------------------------------------------------------------------- 
FUNCTION_BLOCK FB_NovRam EXTENDS FB_Basic IMPLEMENTS I_NovRam
VAR
//**********************************
// Static variables
//**********************************
	_bEnable: BOOL;
	_nDevId: UINT;
	_nMB_Offset: UINT;
	_nMB_Size: UINT;
//**********************************
// Methods variable
//**********************************
	FB_NovRam_M_nEnable_nMBSrc AT %MB0: BYTE;
	FB_NovRam_M_nEnable_nBank: BYTE;
	FB_NovRam_M_nEnable_nCalcSize: UINT;
	FB_NovRam_M_nEnable_iState: UINT;
	FB_NovRam_M_nEnable_fbExecute_R_TRIG: Tc2_Standard.R_TRIG;
	FB_NovRam_M_nEnable_fbExecute_F_TRIG: Tc2_Standard.F_TRIG;
	FB_NovRam_M_nEnable_fbGetDPRAMInfo: Tc2_IoFunctions.FB_GetDPRAMInfo;
	FB_NovRam_M_nEnable_stNovRamAddrInfo: Tc2_IoFunctions.ST_NovRamAddrInfo;
	FB_NovRam_M_nEnable_nArrStatus: ARRAY[1..5] OF UDINT;

	FB_NovRam_M_nRead_fbNovRamReadWriteEx: FB_NovRamReadWriteEx;
	FB_NovRam_M_nRead_iState: UINT;
	FB_NovRam_M_nRead_nBank: BYTE;

	FB_NovRam_M_nWrite_fbNovRamReadWriteEx: FB_NovRamReadWriteEx;
	FB_NovRam_M_nWrite_bReady: BOOL;
	FB_NovRam_M_nWrite_iState: UINT;
	FB_NovRam_M_nWrite_nBank: BYTE;
	FB_NovRam_M_nWrite_pByte: POINTER TO BYTE;
	FB_NovRam_M_nWrite_pCard: POINTER TO BYTE;
END_VAR

//	The result of the method is an unsigned double integer
//	0 = idle 
//	1 = coupled
//	2 = starting
//	3 = running
//	4 = aborted
// 	5 = no hardware connected
// 	6 = spare
//	7 = pointer or index error
//	8 = mapping error
//	9 = parameter error
//	10 = complete
//	Any other number = ErrorID
METHOD PUBLIC M_nEnable : UDINT
VAR_INPUT
	bExecute: BOOL;
	nDevId: UINT;
	nMB_Offset: UINT;
	nMB_Size: UINT;
END_VAR
//**********************************
// Local variable
//**********************************
THIS^._bEnable:= bExecute;
THIS^._nDevId:= nDevId;
THIS^._nMB_Offset:= nMB_Offset;
THIS^._nMB_Size:= nMB_Size;

//**********************************
// Reset
//**********************************
IF _bReset THEN
	IF _bError THEN
		FB_NovRam_M_nEnable_iState:= 000;
	END_IF
	M_nReset(bExecute:= _bReset);
END_IF

//**********************************
// Wait for execute
//**********************************
FB_NovRam_M_nEnable_fbExecute_R_TRIG(CLK:= bExecute);
FB_NovRam_M_nEnable_fbExecute_F_TRIG(CLK:= bExecute);
IF FB_NovRam_M_nEnable_fbExecute_R_TRIG.Q OR FB_NovRam_M_nEnable_fbExecute_F_TRIG.Q THEN
	FB_NovRam_M_nEnable_iState:= 000;
END_IF


//**********************************
// State maschine
//**********************************
CASE FB_NovRam_M_nEnable_iState OF
	
	000:	// Init
			_bReady:= FALSE; 
			FB_NovRam_M_nEnable_fbGetDPRAMInfo(bExecute:= FALSE); 
			IF M_nRead(bExecute:= FALSE) = cIDLE AND M_nWrite(bExecute:= FALSE) = cIDLE THEN
				FB_NovRam_M_nEnable_iState:= FB_NovRam_M_nEnable_iState +1;
			END_IF
	
	001:	// Wait for execute 
			IF bExecute THEN
				FB_NovRam_M_nEnable_iState:= FB_NovRam_M_nEnable_iState +1;
			END_IF
		
	002:	// Check parameter	
			M_nEnable:= cRUNNING;	
			IF _nDevId > 0 AND (nMB_Offset MOD 4 = 0) AND _nMB_Size > 0 AND (_nMB_Size MOD 4 = 0) THEN
				FB_NovRam_M_nEnable_iState:= FB_NovRam_M_nEnable_iState +1;
			ELSE
				M_nEnable:= cPARAMETER_ERROR;	
			END_IF	
		
	003:	// Calculate NovRam Size for ARM cpu
			M_nEnable:= cRUNNING;	
			IF (_nMB_Size + nMB_Offset) MOD 4 = 0 THEN
				FB_NovRam_M_nEnable_nCalcSize:= (_nMB_Size + nMB_Offset);
			ELSE
				FB_NovRam_M_nEnable_nCalcSize:= ((_nMB_Size + nMB_Offset) - (_nMB_Size + nMB_Offset MOD 4))+ 4;
			END_IF
			FB_NovRam_M_nEnable_iState:= FB_NovRam_M_nEnable_iState +1;
		
	004:	// Read NovRam size 
			M_nEnable:= cRUNNING;	
			FB_NovRam_M_nEnable_fbGetDPRAMInfo(
				nDevId:= _nDevId, 
				bExecute:= TRUE, 
				tTimeOut:= Tc2_System.DEFAULT_ADS_TIMEOUT, 
				bBusy=> , 
				bError=> , 
				nErrid=> , 
				stInfo=> FB_NovRam_M_nEnable_stNovRamAddrInfo);
	
			// Error
			IF FB_NovRam_M_nEnable_fbGetDPRAMInfo.bError THEN
				M_nError(nErrorID:= FB_NovRam_M_nEnable_fbGetDPRAMInfo.nErrId);
				M_nEnable:= FB_NovRam_M_nEnable_fbGetDPRAMInfo.nErrId;
			ELSE
				// Done
				IF NOT FB_NovRam_M_nEnable_fbGetDPRAMInfo.bBusy THEN
					FB_NovRam_M_nEnable_fbGetDPRAMInfo(bExecute:= FALSE); 
					FB_NovRam_M_nEnable_iState:= FB_NovRam_M_nEnable_iState +1;
				END_IF
			END_IF	
		
	005:	// Check max NovRam size
			M_nEnable:= cRUNNING;	
			IF FB_NovRam_M_nEnable_nCalcSize > ((FB_NovRam_M_nEnable_stNovRamAddrInfo.iCardMemSize/2) - 2) THEN
				FB_NovRam_M_nEnable_nCalcSize:= UDINT_TO_UINT(FB_NovRam_M_nEnable_stNovRamAddrInfo.iCardMemSize/2);
				FB_NovRam_M_nEnable_nCalcSize:= FB_NovRam_M_nEnable_nCalcSize - 4;
			END_IF
			FB_NovRam_M_nEnable_iState:= FB_NovRam_M_nEnable_iState +1;
	
	006:	// Read
			M_nEnable:= cRUNNING;	
			FB_NovRam_M_nEnable_nArrStatus[1]:= M_nRead(bExecute:= TRUE);
	
			// Error
			IF FB_NovRam_M_nEnable_nArrStatus[1] > cCOMPLETE THEN
				M_nError(nErrorID:= FB_NovRam_M_nEnable_nArrStatus[1]);
				M_nEnable:= FB_NovRam_M_nEnable_nArrStatus[1];
			ELSE
				// Done
				IF FB_NovRam_M_nEnable_nArrStatus[1] = cCOMPLETE THEN
					M_nRead(bExecute:= FALSE);
					FB_NovRam_M_nEnable_iState:= FB_NovRam_M_nEnable_iState +1;
				END_IF
			END_IF
			
	007:	// Write
			M_nEnable:= cRUNNING;	
			FB_NovRam_M_nEnable_nArrStatus[2]:= M_nWrite(bExecute:= TRUE);
			
			// Error
			IF FB_NovRam_M_nEnable_nArrStatus[2] > cCOMPLETE THEN
				M_nError(nErrorID:= FB_NovRam_M_nEnable_nArrStatus[2]);
				M_nEnable:= FB_NovRam_M_nEnable_nArrStatus[2];
			ELSE
				// Done
				IF FB_NovRam_M_nEnable_nArrStatus[2] = cCOMPLETE THEN
					M_nWrite(bExecute:= FALSE);
					FB_NovRam_M_nEnable_iState:= FB_NovRam_M_nEnable_iState +1;
				END_IF
			END_IF
	
	008:	// Done
			M_nEnable:= cCOMPLETE;	
			M_nWrite(bExecute:= TRUE);
			_bReady:= TRUE; 

ELSE
	FB_NovRam_M_nEnable_iState:= 000;
END_CASE
END_METHOD

//	The result of the method is an unsigned double integer
//	0 = idle 
//	1 = coupled
//	2 = starting
//	3 = running
//	4 = aborted
// 	5 = no hardware connected
// 	6 = spare
//	7 = pointer or index error
//	8 = mapping error
//	9 = parameter error
//	10 = complete
//	Any other number = ErrorID
METHOD PRIVATE M_nRead : UDINT
VAR_INPUT
	bExecute: BOOL;
END_VAR
//**********************************
// Reset
//**********************************
IF _bReset THEN
	IF _bError THEN
		FB_NovRam_M_nRead_iState:= 000;
	END_IF
END_IF


//**********************************
// State maschine 
//**********************************
CASE FB_NovRam_M_nRead_iState OF

	000: 	// Init 
			FB_NovRam_M_nRead_fbNovRamReadWriteEx(bRead:= FALSE, bWrite:= FALSE);
			FB_NovRam_M_nRead_iState:= FB_NovRam_M_nRead_iState +1;

	001:	// Wait for execute 
			IF bExecute THEN
				FB_NovRam_M_nRead_iState:= FB_NovRam_M_nRead_iState +1;
			END_IF

	002:	// Read databank value 
			M_nRead:= cRUNNING;
			FB_NovRam_M_nRead_fbNovRamReadWriteEx(
				nDevId:= _nDevId,
				bRead:= TRUE,
				bWrite:= FALSE,
				cbSrcLen:= 1,
				cbDestLen:= 1,
				pSrcAddr:= ADR(FB_NovRam_M_nRead_nBank),
				pDestAddr:= ADR(FB_NovRam_M_nRead_nBank),
				nReadOffs:= FB_NovRam_M_nEnable_stNovRamAddrInfo.iCardMemSize -1,
				nWriteOffs:= 0,
				tTimeOut:= T#2s,
				bBusy=> ,
				bError=> ,
				nErrId=> ,
				cbRead=> ,
				cbWrite=> );
	
			// Error	
			IF FB_NovRam_M_nRead_fbNovRamReadWriteEx.bError THEN
				M_nError(nErrorID:= FB_NovRam_M_nRead_fbNovRamReadWriteEx.nErrId);
				M_nRead:= FB_NovRam_M_nRead_fbNovRamReadWriteEx.nErrId;
			ELSE
				// Done
				IF NOT FB_NovRam_M_nRead_fbNovRamReadWriteEx.bBusy AND FB_NovRam_M_nRead_fbNovRamReadWriteEx.cbRead = 1 THEN
					FB_NovRam_M_nRead_fbNovRamReadWriteEx(bRead:= FALSE,	bWrite:= FALSE);
					FB_NovRam_M_nRead_iState:= FB_NovRam_M_nRead_iState +1;
				END_IF
			END_IF
	
	003:	// ReadNovRam data from databank 0 or 1 
			M_nRead:= cRUNNING;
			IF FB_NovRam_M_nRead_nBank = 0 THEN
				FB_NovRam_M_nRead_fbNovRamReadWriteEx(
					nDevId:= _nDevId,
					bRead:= TRUE,
					bWrite:= FALSE,
					cbSrcLen:= FB_NovRam_M_nEnable_nCalcSize,
					cbDestLen:= FB_NovRam_M_nEnable_nCalcSize,
					pSrcAddr:= ADR(FB_NovRam_M_nEnable_nMBSrc),
					pDestAddr:= ADR(FB_NovRam_M_nEnable_nMBSrc),
					nReadOffs:= 0,
					nWriteOffs:= 0,
					tTimeOut:= T#2s,
					bBusy=> ,
					bError=> ,
					nErrId=> ,
					cbRead=> ,
					cbWrite=> );
			ELSE
				FB_NovRam_M_nRead_fbNovRamReadWriteEx(
					nDevId:= _nDevId,
					bRead:= TRUE,
					bWrite:= FALSE,
					cbSrcLen:= FB_NovRam_M_nEnable_nCalcSize,
					cbDestLen:= FB_NovRam_M_nEnable_nCalcSize,
					pSrcAddr:= ADR(FB_NovRam_M_nEnable_nMBSrc),
					pDestAddr:= ADR(FB_NovRam_M_nEnable_nMBSrc),
					nReadOffs:= FB_NovRam_M_nEnable_stNovRamAddrInfo.iCardMemSize / 2,
					nWriteOffs:= 0,
					tTimeOut:= T#2s,
					bBusy=> ,
					bError=> ,
					nErrId=> ,
					cbRead=> ,
					cbWrite=> );
			END_IF
	
			// Error	
			IF FB_NovRam_M_nRead_fbNovRamReadWriteEx.bError THEN
				M_nError(nErrorID:= FB_NovRam_M_nRead_fbNovRamReadWriteEx.nErrId);
				M_nRead:= FB_NovRam_M_nRead_fbNovRamReadWriteEx.nErrId;
			ELSE
				// Done
				IF NOT FB_NovRam_M_nRead_fbNovRamReadWriteEx.bBusy AND FB_NovRam_M_nRead_fbNovRamReadWriteEx.cbRead = FB_NovRam_M_nEnable_nCalcSize THEN
					FB_NovRam_M_nRead_fbNovRamReadWriteEx(bRead:= FALSE,	bWrite:= FALSE);
					FB_NovRam_M_nRead_iState:= FB_NovRam_M_nRead_iState +1;
				END_IF
			END_IF
	
	004:	// Read done 
			M_nRead:= cCOMPLETE;
			IF NOT bExecute THEN
				FB_NovRam_M_nRead_iState:= 000;
			END_IF

ELSE
	FB_NovRam_M_nRead_iState:= 000;
END_CASE
END_METHOD

//	The result of the method is an unsigned double integer
//	0 = idle 
//	1 = coupled
//	2 = starting
//	3 = running
//	4 = aborted
// 	5 = no hardware connected
// 	6 = spare
//	7 = pointer or index error
//	8 = mapping error
//	9 = parameter error
//	10 = complete
//	Any other number = ErrorID
METHOD PRIVATE M_nWrite : UDINT
VAR_INPUT
	bExecute: BOOL;
END_VAR
//**********************************
// Reset
//**********************************
IF _bReset THEN
	IF _bError THEN
		FB_NovRam_M_nWrite_iState:= 000;
	END_IF
END_IF


//**********************************
// State maschine 
//**********************************
CASE FB_NovRam_M_nWrite_iState OF

	000:	// Init
			FB_NovRam_M_nWrite_fbNovRamReadWriteEx(bRead:= FALSE,	bWrite:= FALSE);
			FB_NovRam_M_nWrite_bReady:= FALSE;
			FB_NovRam_M_nWrite_iState:= FB_NovRam_M_nWrite_iState +1;

	001:	// Wait for execute 
			IF bExecute THEN
				FB_NovRam_M_nWrite_iState:= FB_NovRam_M_nWrite_iState +1;
			END_IF

	002:	// Read databank value 
			M_nWrite:= cSTARTING;
			FB_NovRam_M_nWrite_fbNovRamReadWriteEx(
				nDevId:= _nDevId,
				bRead:= TRUE,
				bWrite:= FALSE,
				cbSrcLen:= 1,
				cbDestLen:= 1,
				pSrcAddr:= ADR(FB_NovRam_M_nWrite_nBank),
				pDestAddr:= ADR(FB_NovRam_M_nWrite_nBank),
				nReadOffs:= FB_NovRam_M_nEnable_stNovRamAddrInfo.iCardMemSize -1,
				nWriteOffs:= 0,
				tTimeOut:= T#2s,
				bBusy=> ,
				bError=> ,
				nErrId=> ,
				cbRead=> ,
				cbWrite=> );
	
			// Error
			IF FB_NovRam_M_nWrite_fbNovRamReadWriteEx.bError THEN
				M_nError(nErrorID:= FB_NovRam_M_nWrite_fbNovRamReadWriteEx.nErrId);
				M_nWrite:= FB_NovRam_M_nWrite_fbNovRamReadWriteEx.nErrId;
			ELSE	
				// Done				
				IF FB_NovRam_M_nWrite_fbNovRamReadWriteEx.cbRead = 1 THEN
					FB_NovRam_M_nWrite_fbNovRamReadWriteEx(bRead:= FALSE,	bWrite:= FALSE);
					FB_NovRam_M_nWrite_iState:= FB_NovRam_M_nWrite_iState +1;
				END_IF
			END_IF
		
	003:	// Pointer settings 
			M_nWrite:= cSTARTING;
			FB_NovRam_M_nWrite_pByte:= ADR(FB_NovRam_M_nWrite_nBank);
			FB_NovRam_M_nWrite_pCard:= FB_NovRam_M_nEnable_stNovRamAddrInfo.pCardAddress + FB_NovRam_M_nEnable_stNovRamAddrInfo.iCardMemSize -1;
			FB_NovRam_M_nWrite_iState:= FB_NovRam_M_nWrite_iState +1;
		
	004:	// Write ready 
			M_nWrite:= cCOMPLETE;
			FB_NovRam_M_nWrite_bReady:= TRUE;
			IF NOT bExecute THEN
				FB_NovRam_M_nWrite_iState:= 000;
			END_IF
		
ELSE
	FB_NovRam_M_nWrite_iState:= 000;
END_CASE


// Write data to databank 0 or 1 
IF bExecute AND FB_NovRam_M_nWrite_bReady THEN
	IF FB_NovRam_M_nWrite_nBank = 1 THEN
		FB_NovRam_M_nWrite_nBank:= 0;
		MEMCPY(destAddr:= FB_NovRam_M_nEnable_stNovRamAddrInfo.pCardAddress, srcAddr:= ADR(FB_NovRam_M_nEnable_nMBSrc) + _nMB_Offset, n:= FB_NovRam_M_nEnable_nCalcSize);
		FB_NovRam_M_nWrite_pCard^:= FB_NovRam_M_nWrite_pByte^;
	ELSE
		FB_NovRam_M_nWrite_nBank:= 1;
		MEMCPY(destAddr:= FB_NovRam_M_nEnable_stNovRamAddrInfo.pCardAddress + (FB_NovRam_M_nEnable_stNovRamAddrInfo.iCardMemSize/2), srcAddr:= ADR(FB_NovRam_M_nEnable_nMBSrc) + _nMB_Offset, n:= FB_NovRam_M_nEnable_nCalcSize);
		FB_NovRam_M_nWrite_pCard^:= FB_NovRam_M_nWrite_pByte^;
	END_IF
END_IF
END_METHOD

END_FUNCTION_BLOCK

// POUs/SYSTEM/POUs/FBs/Persistent/ITFs/I_WritePersistentData
INTERFACE I_WritePersistentData EXTENDS I_Basic

//	The result of the method is an unsigned double integer
//	0 = idle 
//	1 = coupled
//	2 = starting
//	3 = running
//	4 = aborted
// 	5 = no hardware connected
//  6 = Spare
//	7 = pointer or index error
//	8 = mapping error
//	9 = parameter error
//	10 = complete
//	Any other number = ErrorID
METHOD PUBLIC M_n1_Second_UPS : UDINT
VAR_INPUT
	bExecute: BOOL;
END_VAR
END_METHOD

//	The result of the method is an unsigned double integer
//	0 = idle 
//	1 = coupled
//	2 = starting
//	3 = running
//	4 = aborted
// 	5 = no hardware connected
//  6 = Spare
//	7 = pointer or index error
//	8 = mapping error
//	9 = parameter error
//	10 = complete
//	Any other number = ErrorID
METHOD M_nEnable : UDINT
VAR_INPUT
	bExecute: BOOL;
	tLogTimePuls: TIME;
END_VAR
END_METHOD

//	The result of the method is an unsigned double integer
//	0 = idle 
//	1 = coupled
//	2 = starting
//	3 = running
//	4 = aborted
// 	5 = no hardware connected
//  6 = Spare
//	7 = pointer or index error
//	8 = mapping error
//	9 = parameter error
//	10 = complete
//	Any other number = ErrorID
METHOD M_nWrite : UDINT
VAR_INPUT
	bExecute: BOOL;
END_VAR
END_METHOD

PROPERTY PUBLIC P_bBusy : BOOL
GET
END_GET
END_PROPERTY

PROPERTY PUBLIC P_bPowerFailDetect : BOOL
GET
END_GET
END_PROPERTY

PROPERTY PUBLIC P_eSUPS_Mode : Tc2_SUPS.E_S_UPS_Mode
SET
END_SET
END_PROPERTY

PROPERTY PUBLIC P_nWriteCNT : UDINT
GET
END_GET
END_PROPERTY

END_INTERFACE

// POUs/SYSTEM/POUs/FBs/Persistent/FB_WritePersistentData
//------------------------------------------------------------------------------------------
//                                                                                        	
//***************************** Beckhoff TwinCAT Examples **********************************
//                                                                                        	
//************************************* WARNING ********************************************
// This program is only an example. If it is used as a control program in any real        	
// application, Beckhoff is not responsible for any malfunction, loss or damage           	
// which could arise by using this program!                                               	
//                                                                                        	
//*************************************  Program Info. *************************************
//                                                                                        	
// PLC program name:       	FB_WritePersistentData (FB)                                          	
// Hardware platform:      	TwinCat v3.1.4022				                          		                                  	
//                                                                                        	
// ======================================================================================== 
//         Version       Date                        Remarks                              	
// ======================================================================================== 
//         3.1           27 feb 2018                 First release of this example        	
// ======================================================================================== 
//                                                                                        	
//******************************* Aims OF this PLC PROGRAM *********************************
//                                                                                        	
// Write persistent data file				 			                                      	
//																	                      	
//                                                                                        	
//----------------------------------------------------------------------------------------- 
FUNCTION_BLOCK FB_WritePersistentData EXTENDS FB_Basic IMPLEMENTS I_WritePersistentData
VAR
//**************************
// Static variables
//**************************
	_bFirstBoot: BOOL := TRUE;
	_nAdsPort: UINT;
	_bPowerFailDetect: BOOL;
	_fbWritePersistentData: Tc2_Utilities.FB_WritePersistentData;
	_nWriteCNT: UDINT;
	_eUpsMode: Tc2_SUPS.E_S_UPS_Mode;
	
//**************************
// Property variables
//**************************
	_bBusy: BOOL;	
	
//**************************
// Methods variable
//**************************

	FB_WritePersistentData_M_nEnable_iState: INT;
	FB_WritePersistentData_M_nEnable_fbExecute_R_TRIG: R_TRIG;
	FB_WritePersistentData_M_nEnable_fbReset_R_TRIG: R_TRIG;
	FB_WritePersistentData_M_nEnable_fbStartDelay_TON: TON;
	FB_WritePersistentData_M_nEnable_fbLogTimePuls_TON: TON;
	
	FB_WritePersistentData_M_nWrite_iState: INT;
	FB_WritePersistentData_M_nWrite_fbExecute_R_TRIG: R_TRIG;
	FB_WritePersistentData_M_nWrite_fbReset_R_TRIG: R_TRIG;
	
	FB_WritePersistentData_M_n1_Second_UPS_iState: INT;
	FB_WritePersistentData_M_n1_Second_UPS_bIs_CB3011: BOOL;
	FB_WritePersistentData_M_n1_Second_UPS_bIs_CX9020_U900: BOOL;
	FB_WritePersistentData_M_n1_Second_UPS_bIs_CX50x0: BOOL;
	FB_WritePersistentData_M_n1_Second_UPS_bIs_CX51x0: BOOL;
	FB_WritePersistentData_M_n1_Second_UPS_bReady: BOOL;
	FB_WritePersistentData_M_n1_Second_UPS_fb_S_UPS_CB3011: Tc2_SUPS.FB_S_UPS_CB3011; 
	FB_WritePersistentData_M_n1_Second_UPS_fb_S_UPS_CX9020_U900: Tc2_SUPS.FB_S_UPS_CX9020_U900; 
	FB_WritePersistentData_M_n1_Second_UPS_fb_S_UPS_CX50x0: Tc2_SUPS.FB_S_UPS;
	FB_WritePersistentData_M_n1_Second_UPS_fb_S_UPS_CX51x0: Tc2_SUPS.FB_S_UPS_CX51x0;
	FB_WritePersistentData_M_n1_Second_UPS_stDeviceIdentificationEx: Tc2_Utilities.ST_DeviceIdentificationEx;
	FB_WritePersistentData_M_n1_Second_UPS_fb_GetDeviceIdentificationEx: Tc2_Utilities.FB_GetDeviceIdentificationEx;
	
END_VAR

//	The result of the method is an unsigned double integer
//	0 = idle 
//	1 = coupled
//	2 = starting
//	3 = running
//	4 = aborted
// 	5 = no hardware connected
// 	6 = spare
//	7 = pointer or index error
//	8 = mapping error
//	9 = parameter error
//	10 = complete
//	Any other number = ErrorID
METHOD PUBLIC M_n1_Second_UPS : UDINT
VAR_INPUT
	bExecute: BOOL;
END_VAR
_bPowerFailDetect:= FALSE;

// Check normal backup is not running
IF NOT _bBusy THEN
	IF FB_WritePersistentData_M_n1_Second_UPS_bReady THEN
		
		// Update CB3011 UPS
		IF FB_WritePersistentData_M_n1_Second_UPS_bIs_CB3011 THEN
			FB_WritePersistentData_M_n1_Second_UPS_fb_S_UPS_CB3011(
				sNetID:= , 
				iPLCPort:= TwinCAT_SystemInfoVarList._AppInfo.AdsPort, 
				tTimeout:= , 
				eUpsMode:= _eUpsMode, 
				ePersistentMode:= , 
				tRecoverTime:= , 
				bPowerFailDetect=> _bPowerFailDetect, 
				eState=> );
		END_IF
		
		// Update CX9020-U900 UPS
		IF FB_WritePersistentData_M_n1_Second_UPS_bIs_CX9020_U900 THEN
			FB_WritePersistentData_M_n1_Second_UPS_fb_S_UPS_CX9020_U900(
				sNetID:= , 
				iPLCPort:= TwinCAT_SystemInfoVarList._AppInfo.AdsPort, 
				tTimeout:= , 
				eUpsMode:= _eUpsMode, 
				ePersistentMode:= , 
				tRecoverTime:= , 
				bPowerFailDetect=> _bPowerFailDetect, 
				eState=> );
		END_IF
		
		// Update CX50x0 UPS
		IF FB_WritePersistentData_M_n1_Second_UPS_bIs_CX50x0 THEN
			FB_WritePersistentData_M_n1_Second_UPS_fb_S_UPS_CX50x0(
				sNetID:= , 
				iPLCPort:= TwinCAT_SystemInfoVarList._AppInfo.AdsPort, 
				iUPSPort:= , 
				tTimeout:= , 
				eUpsMode:= _eUpsMode, 
				ePersistentMode:= , 
				tRecoverTime:= , 
				bPowerFailDetect=> _bPowerFailDetect, 
				eState=> );
		END_IF
		
		// Update CX51x0 UPS
		IF FB_WritePersistentData_M_n1_Second_UPS_bIs_CX51x0 THEN
			FB_WritePersistentData_M_n1_Second_UPS_fb_S_UPS_CX51x0(
				sNetID:= , 
				iPLCPort:= TwinCAT_SystemInfoVarList._AppInfo.AdsPort, 
				iUPSPort:= , 
				tTimeout:= , 
				eUpsMode:= _eUpsMode, 
				ePersistentMode:= , 
				tRecoverTime:= , 
				bPowerFailDetect=> _bPowerFailDetect, 
				eState=> );
		END_IF
	
	END_IF
END_IF

	
//**********************************
// Reset 
//**********************************
IF _bReset THEN
	IF _bError THEN	
		FB_WritePersistentData_M_n1_Second_UPS_iState:= 000;
	END_IF	
END_IF


//**********************************
// State maschine
//**********************************
CASE FB_WritePersistentData_M_n1_Second_UPS_iState OF
	
	000:	// Wait for execute and start delay
			FB_WritePersistentData_M_n1_Second_UPS_bReady:= FALSE;
			IF bExecute THEN
				FB_WritePersistentData_M_n1_Second_UPS_iState:= FB_WritePersistentData_M_n1_Second_UPS_iState +1;
			END_IF	

	001:	// Get data	
			M_n1_Second_UPS:= cRUNNING;
			FB_WritePersistentData_M_n1_Second_UPS_fb_GetDeviceIdentificationEx(bExecute:= FALSE); 
			FB_WritePersistentData_M_n1_Second_UPS_fb_GetDeviceIdentificationEx(
				bExecute:= TRUE, 
				tTimeout:= Tc2_System.DEFAULT_ADS_TIMEOUT, 
				sNetId:= '', 
				bBusy=> , 
				bError=> , 
				nErrorID=> , 
				stDevIdent=> FB_WritePersistentData_M_n1_Second_UPS_stDeviceIdentificationEx);
	
			FB_WritePersistentData_M_n1_Second_UPS_iState:= FB_WritePersistentData_M_n1_Second_UPS_iState +1;
	
	002:	// Get data done
			M_n1_Second_UPS:= cRUNNING;
			FB_WritePersistentData_M_n1_Second_UPS_fb_GetDeviceIdentificationEx(bExecute:= FALSE, stDevIdent=> FB_WritePersistentData_M_n1_Second_UPS_stDeviceIdentificationEx);
			IF FB_WritePersistentData_M_n1_Second_UPS_fb_GetDeviceIdentificationEx.bError THEN
				M_nError(nErrorID:= FB_WritePersistentData_M_n1_Second_UPS_fb_GetDeviceIdentificationEx.nErrorID);
				M_n1_Second_UPS:= FB_WritePersistentData_M_n1_Second_UPS_fb_GetDeviceIdentificationEx.nErrorID;
			ELSE
				// Done
				IF NOT FB_WritePersistentData_M_n1_Second_UPS_fb_GetDeviceIdentificationEx.bBusy THEN
					FB_WritePersistentData_M_n1_Second_UPS_iState:= FB_WritePersistentData_M_n1_Second_UPS_iState +1;
				END_IF	
			END_IF
		
	003:	// Check 1s UPS device type
			M_n1_Second_UPS:= cRUNNING;
			FB_WritePersistentData_M_n1_Second_UPS_bIs_CB3011:= Tc2_Standard.MID(FB_WritePersistentData_M_n1_Second_UPS_stDeviceIdentificationEx.strHardwareModel, 5, 1) = 'CB3011';
			FB_WritePersistentData_M_n1_Second_UPS_bIs_CX9020_U900:= Tc2_Standard.MID(FB_WritePersistentData_M_n1_Second_UPS_stDeviceIdentificationEx.strHardwareModel, 11, 1) = 'CX9020-U900';
			FB_WritePersistentData_M_n1_Second_UPS_bIs_CX50x0:= Tc2_Standard.MID(FB_WritePersistentData_M_n1_Second_UPS_stDeviceIdentificationEx.strHardwareModel, 2, 1) = '50';
			FB_WritePersistentData_M_n1_Second_UPS_bIs_CX51x0:= Tc2_Standard.MID(FB_WritePersistentData_M_n1_Second_UPS_stDeviceIdentificationEx.strHardwareModel, 4, 1) = 'CX51';
		
			// 1s UPS hardware connected
			IF FB_WritePersistentData_M_n1_Second_UPS_bIs_CB3011 THEN
				FB_WritePersistentData_M_n1_Second_UPS_iState:= FB_WritePersistentData_M_n1_Second_UPS_iState +2;
			ELSE
				IF FB_WritePersistentData_M_n1_Second_UPS_bIs_CX9020_U900 THEN
					FB_WritePersistentData_M_n1_Second_UPS_iState:= FB_WritePersistentData_M_n1_Second_UPS_iState +2;
				ELSE
					IF FB_WritePersistentData_M_n1_Second_UPS_bIs_CX50x0 THEN
						FB_WritePersistentData_M_n1_Second_UPS_iState:= FB_WritePersistentData_M_n1_Second_UPS_iState +2;
					ELSE
						IF FB_WritePersistentData_M_n1_Second_UPS_bIs_CX51x0 THEN
							FB_WritePersistentData_M_n1_Second_UPS_iState:= FB_WritePersistentData_M_n1_Second_UPS_iState +2;
						ELSE
							FB_WritePersistentData_M_n1_Second_UPS_iState:= FB_WritePersistentData_M_n1_Second_UPS_iState +1;
						END_IF
					END_IF
				END_IF	
			END_IF

	004:	// No 1sec UPS hardware connected	
			IF bExecute THEN
				M_n1_Second_UPS:= cNO_HARDWARE_CONNECTED;
			ELSE
				FB_WritePersistentData_M_n1_Second_UPS_iState:= 000;
			END_IF	
	
	005:	// Wait not Execute
			M_n1_Second_UPS:= cCOMPLETE;
			FB_WritePersistentData_M_n1_Second_UPS_bReady:= TRUE;
			IF NOT bExecute THEN
				FB_WritePersistentData_M_n1_Second_UPS_iState:= 000;
			END_IF	

ELSE
	FB_WritePersistentData_M_n1_Second_UPS_iState:= 000;
END_CASE
END_METHOD

//	The result of the method is an unsigned double integer
//	0 = idle 
//	1 = coupled
//	2 = starting
//	3 = running
//	4 = aborted
// 	5 = no hardware connected
// 	6 = spare
//	7 = pointer or index error
//	8 = mapping error
//	9 = parameter error
//	10 = complete
//	Any other number = ErrorID
METHOD PUBLIC M_nEnable : UDINT
VAR_INPUT
	bExecute: BOOL;
	tLogTimePuls: TIME;
END_VAR
// Local variable
THIS^._nAdsPort:= TwinCAT_SystemInfoVarList._AppInfo.AdsPort;

//**********************************
// Reset 
//**********************************
IF _bReset THEN
	IF _bError THEN	
		FB_WritePersistentData_M_nEnable_iState:= 000;
	END_IF	
	M_nReset(bExecute:= _bReset);
END_IF

// Power fail
FB_WritePersistentData_M_nEnable_fbReset_R_TRIG(CLK:= _bPowerFailDetect, Q=> );
IF FB_WritePersistentData_M_nEnable_fbReset_R_TRIG.Q THEN
	FB_WritePersistentData_M_nEnable_iState:= 000;
END_IF

// Startup delay
FB_WritePersistentData_M_nEnable_fbStartDelay_TON(IN:= TRUE, PT:= T#15S);

// LogTtime puls
IF FB_WritePersistentData_M_nEnable_fbStartDelay_TON.Q THEN
	FB_WritePersistentData_M_nEnable_fbLogTimePuls_TON(IN:= bExecute AND tLogTimePuls > T#0MS AND NOT FB_WritePersistentData_M_nEnable_fbLogTimePuls_TON.Q, PT:= tLogTimePuls);
ELSE
	FB_WritePersistentData_M_nEnable_fbLogTimePuls_TON(IN:= FALSE);
END_IF	

//**********************************
// Wait for execute
//**********************************
IF FB_WritePersistentData_M_nEnable_fbStartDelay_TON.Q THEN
	FB_WritePersistentData_M_nEnable_fbExecute_R_TRIG(CLK:= (_bFirstBoot OR FB_WritePersistentData_M_nEnable_fbLogTimePuls_TON.Q) AND NOT _bPowerFailDetect);
	IF FB_WritePersistentData_M_nEnable_fbExecute_R_TRIG.Q THEN
		FB_WritePersistentData_M_nEnable_iState:= 001;
	END_IF
ELSE
	FB_WritePersistentData_M_nEnable_fbExecute_R_TRIG(CLK:= FALSE);
	FB_WritePersistentData_M_nEnable_iState:= 000;
END_IF


//**********************************
// Main sequence
//**********************************
CASE FB_WritePersistentData_M_nEnable_iState OF

	000:	// Do nothing
			IF _bError THEN
				M_nEnable:= _nErrorID;
			ELSE
				IF bExecute THEN
					IF FB_WritePersistentData_M_nEnable_fbStartDelay_TON.Q THEN
						M_nEnable:= cCOMPLETE;
					ELSE
						M_nEnable:= cSTARTING;
					END_IF
				END_IF	
			END_IF

	001:	// Init
			M_nEnable:= cSTARTING;
			_fbWritePersistentData.PORT:= _nAdsPort;
			_fbWritePersistentData.TMOUT:= Tc2_System.DEFAULT_ADS_TIMEOUT;
			FB_WritePersistentData_M_nEnable_iState:= FB_WritePersistentData_M_nEnable_iState +1;

	002:	// Running
			M_nEnable:= cSTARTING;
			IF _fbWritePersistentData.BUSY THEN
				FB_WritePersistentData_M_nEnable_iState:= FB_WritePersistentData_M_nEnable_iState +3;
			ELSE
				FB_WritePersistentData_M_nEnable_iState:= FB_WritePersistentData_M_nEnable_iState +1;
			END_IF
			
	003:	// Init
			M_nEnable:= cSTARTING;
			_fbWritePersistentData.START:= FALSE; 
			FB_WritePersistentData_M_nEnable_iState:= FB_WritePersistentData_M_nEnable_iState +1;

	004:	// Start
			M_nEnable:= cSTARTING;
			_fbWritePersistentData.START:= TRUE; 
			FB_WritePersistentData_M_nEnable_iState:= FB_WritePersistentData_M_nEnable_iState +1;

	005:	// Write persistent data - Done
			M_nEnable:= cSTARTING;
		
			// Error handling
			IF _fbWritePersistentData.ERR THEN
				M_nError(nErrorID:= _fbWritePersistentData.ERRID);	
				M_nEnable:= _fbWritePersistentData.ERRID;
			ELSE
				// Done
				IF NOT _fbWritePersistentData.BUSY THEN
					IF _bFirstBoot THEN
						_fbWritePersistentData.START:= FALSE; 
						FB_WritePersistentData_M_nEnable_iState:= FB_WritePersistentData_M_nEnable_iState +1;
					ELSE
						_nWriteCNT:= _nWriteCNT +1;
						_fbWritePersistentData.START:= FALSE; 
						FB_WritePersistentData_M_nEnable_iState:= 100;
					END_IF
				END_IF	
			END_IF

	006:	// Init
			M_nEnable:= cSTARTING;
			_fbWritePersistentData.START:= FALSE; 
			FB_WritePersistentData_M_nEnable_iState:= FB_WritePersistentData_M_nEnable_iState +1;

	007:	// Start
			M_nEnable:= cSTARTING;
			_fbWritePersistentData.START:= TRUE; 
			FB_WritePersistentData_M_nEnable_iState:= FB_WritePersistentData_M_nEnable_iState +1;
			
	008:	// Write persistent data - Done
			M_nEnable:= cSTARTING;
		
			// Error handling
			IF _fbWritePersistentData.ERR THEN
				M_nError(nErrorID:= _fbWritePersistentData.ERRID);	
				M_nEnable:= _fbWritePersistentData.ERRID;
			ELSE
				// Done
				IF NOT _fbWritePersistentData.BUSY THEN
					_nWriteCNT:= _nWriteCNT +1;
					_fbWritePersistentData.START:= FALSE; 
					FB_WritePersistentData_M_nEnable_iState:= 100;
				END_IF	
			END_IF
	
	100:	// Done
			M_nEnable:= cCOMPLETE;
			_bFirstBoot:= FALSE;
			FB_WritePersistentData_M_nEnable_iState:= 000;

ELSE
	FB_WritePersistentData_M_nEnable_iState:= 000;	
END_CASE


// Proporty update
IF NOT _bError AND FB_WritePersistentData_M_nEnable_fbStartDelay_TON.Q AND NOT _bPowerFailDetect THEN
	_bReady:= TRUE; 
ELSE
	_bReady:= FALSE; 
END_IF

// Status update
_fbWritePersistentData(TMOUT:= T#30S); 
_bBusy:= _fbWritePersistentData.BUSY;
END_METHOD

//	The result of the method is an unsigned double integer
//	0 = idle 
//	1 = coupled
//	2 = starting
//	3 = running
//	4 = aborted
// 	5 = no hardware connected
// 	6 = spare
//	7 = pointer or index error
//	8 = mapping error
//	9 = parameter error
//	10 = complete
//	Any other number = ErrorID
METHOD PUBLIC M_nWrite : UDINT
VAR_INPUT
	bExecute: BOOL;
END_VAR
//**********************************
// Reset 
//**********************************
IF _bReset THEN
	IF _bError THEN	
		FB_WritePersistentData_M_nWrite_iState:= 000;
	END_IF	
END_IF

// Power fail
FB_WritePersistentData_M_nWrite_fbReset_R_TRIG(CLK:= _bPowerFailDetect, Q=> );
IF FB_WritePersistentData_M_nWrite_fbReset_R_TRIG.Q THEN
	FB_WritePersistentData_M_nWrite_iState:= 000;
END_IF

//**********************************
// Wait for execute
//**********************************
IF _bReady THEN
	FB_WritePersistentData_M_nWrite_fbExecute_R_TRIG(CLK:= bExecute AND NOT _bPowerFailDetect);
	IF FB_WritePersistentData_M_nWrite_fbExecute_R_TRIG.Q THEN
		FB_WritePersistentData_M_nWrite_iState:= 001;
	END_IF
ELSE
	FB_WritePersistentData_M_nWrite_fbExecute_R_TRIG(CLK:= FALSE);
	FB_WritePersistentData_M_nWrite_iState:= 000;
END_IF


//**********************************
// Main sequence
//**********************************
CASE FB_WritePersistentData_M_nWrite_iState OF

	000:	// Do nothing
	
	001:	// Running
			M_nWrite:= cRUNNING;
			IF _bBusy THEN
				FB_WritePersistentData_M_nWrite_iState:= FB_WritePersistentData_M_nWrite_iState +1;
			ELSE
				FB_WritePersistentData_M_nWrite_iState:= FB_WritePersistentData_M_nWrite_iState +2;
			END_IF

	002:	// Write persistent done
			M_nWrite:= cRUNNING;
			IF NOT _bBusy THEN
				_fbWritePersistentData.START:= FALSE; 
				FB_WritePersistentData_M_nWrite_iState:= 100;
			END_IF
			
	003:	// Init
			M_nWrite:= cRUNNING;
			_fbWritePersistentData.START:= FALSE; 
			FB_WritePersistentData_M_nWrite_iState:= FB_WritePersistentData_M_nWrite_iState +1;

	004:	// Start
			M_nWrite:= cRUNNING;
			_fbWritePersistentData.START:= TRUE; 
			FB_WritePersistentData_M_nWrite_iState:= FB_WritePersistentData_M_nWrite_iState +1;

	005:	// Write persistent data - Done
			M_nWrite:= cRUNNING;
		
			// Error handling
			IF _fbWritePersistentData.ERR THEN
				M_nError(nErrorID:= _fbWritePersistentData.ERRID);	
				M_nWrite:= _fbWritePersistentData.ERRID;
			ELSE
				// Done
				IF NOT _bBusy THEN
					_nWriteCNT:= _nWriteCNT +1;
					_fbWritePersistentData.START:= FALSE; 	
					FB_WritePersistentData_M_nWrite_iState:= 100;
				END_IF	
			END_IF
	
	100:	// Done
			M_nWrite:= cCOMPLETE;
			IF NOT bExecute THEN
				FB_WritePersistentData_M_nWrite_iState:= 000;	
			END_IF	
	
ELSE
	FB_WritePersistentData_M_nWrite_iState:= 000;	
END_CASE
END_METHOD

PROPERTY PUBLIC P_bBusy : BOOL
GET
P_bBusy:= _bBusy;
END_GET
END_PROPERTY

PROPERTY PUBLIC P_bPowerFailDetect : BOOL
GET
P_bPowerFailDetect:= _bPowerFailDetect;
END_GET
END_PROPERTY

PROPERTY PUBLIC P_eSUPS_Mode : Tc2_SUPS.E_S_UPS_Mode
SET
_eUpsMode:= P_eSUPS_Mode;
END_SET
END_PROPERTY

PROPERTY PUBLIC P_nWriteCNT : UDINT
GET
P_nWriteCNT:= _nWriteCNT;
END_GET
END_PROPERTY

END_FUNCTION_BLOCK

// POUs/SYSTEM/POUs/FBs/System/ITFs/I_System
INTERFACE I_System EXTENDS I_Basic

//	The result of the method is an unsigned double integer
//	0 = idle 
//	1 = coupled
//	2 = starting
//	3 = running
//	4 = aborted
// 	5 = no hardware connected
//  6 = Spare
//	7 = pointer or index error
//	8 = mapping error
//	9 = parameter error
//	10 = complete
//	Any other number = ErrorID
METHOD PUBLIC M_nCerHost : UDINT
VAR_INPUT
	bEnable: BOOL;
	bDisable: BOOL;
END_VAR
END_METHOD

//	The result of the method is an unsigned double integer
//	0 = idle 
//	1 = coupled
//	2 = starting
//	3 = running
//	4 = aborted
// 	5 = no hardware connected
//  6 = Spare
//	7 = pointer or index error
//	8 = mapping error
//	9 = parameter error
//	10 = complete
//	Any other number = ErrorID
METHOD PUBLIC M_nEnable : UDINT
VAR_INPUT
END_VAR
END_METHOD

METHOD PUBLIC M_nGetTimeStampInMs : ULINT
VAR_INPUT
END_VAR
END_METHOD

PROPERTY PUBLIC P_bIs_ARM : BOOL
GET
END_GET
END_PROPERTY

PROPERTY PUBLIC P_bIs_CE_Device : BOOL
GET
END_GET
END_PROPERTY

PROPERTY PUBLIC P_bIs_x64 : BOOL
GET
END_GET
END_PROPERTY

PROPERTY PUBLIC P_bIs_x86 : BOOL
GET
END_GET
END_PROPERTY

PROPERTY PUBLIC P_nAdsPort : UINT
GET
END_GET
END_PROPERTY

PROPERTY PUBLIC P_nCycleTime : UDINT
GET
END_GET
END_PROPERTY

PROPERTY PUBLIC P_stDeviceIdentificationEx : Tc2_Utilities.ST_DeviceIdentificationEx
GET
END_GET
END_PROPERTY

PROPERTY PUBLIC P_sTwinCAT_Version : STRING
GET
END_GET
END_PROPERTY

END_INTERFACE

// POUs/SYSTEM/POUs/FBs/System/FB_System
//------------------------------------------------------------------------------------------
//                                                                                        	
//***************************** Beckhoff TwinCAT Examples **********************************
//                                                                                        	
//************************************* WARNING ********************************************
// This program is only an example. If it is used as a control program in any real        	
// application, Beckhoff is not responsible for any malfunction, loss or damage           	
// which could arise by using this program!                                               	
//                                                                                        	
//*************************************  Program Info. *************************************
//                                                                                        	
// PLC program name:       	FB_System (FB)               	                           	
// Hardware platform:      	TwinCat v3.1.4022				                          		                                  	
//                                                                                        	
// ======================================================================================== 
//         Version       Date                        Remarks                              	
// ======================================================================================== 
//         3.1           27 feb 2018                 First release of this example  
//         3.2.1.1       09 march 2018                 First release of this example        	
// ======================================================================================== 
//                                                                                        	
//******************************* Aims OF this PLC PROGRAM *********************************
//                                                                                        	
//	TwinCAT device info																	                      	
//                                                                                        	
//----------------------------------------------------------------------------------------- 
FUNCTION_BLOCK FB_System EXTENDS FB_Basic IMPLEMENTS I_System
VAR
{attribute 'hide'}
	pInternPointer: POINTER TO INT;
END_VAR
VAR
//**************************
// Property variables
//**************************
	_bIs_ARM: BOOL;
	_stDeviceIdentificationEx: Tc2_Utilities.ST_DeviceIdentificationEx;
	_sTwinCAT_Version: STRING(20);

	
//**********************************
// Methods variable
//**********************************
	FB_System_M_nEnable_iState: INT;
	FB_System_M_nEnable_bDone: BOOL; 
	FB_System_M_nEnable_arrUINT: ARRAY[1..4] OF UINT;
	FB_System_M_nEnable_stDeviceIdentificationEx: Tc2_Utilities.ST_DeviceIdentificationEx;
	FB_System_M_nEnable_fb_GetDeviceIdentificationEx: Tc2_Utilities.FB_GetDeviceIdentificationEx;
	FB_System_M_nEnable_fbADSREAD: Tc2_System.ADSREAD;
	
	FB_System_M_nCerHost_iState: INT;
	FB_System_M_nCerHost_sValue: STRING;
	FB_System_M_nCerHost_fbEnable_R_TRIG: Tc2_Standard.R_TRIG;
	FB_System_M_nCerHost_fbDisable_R_TRIG: Tc2_Standard.R_TRIG;
	FB_System_M_nCerHost_fbRegSetValue: Tc2_Utilities.FB_RegSetValue;
	FB_System_M_nCerHost_fbNT_Reboot: Tc2_Utilities.NT_Reboot;
END_VAR

//	The result of the method is an unsigned double integer
//	0 = idle 
//	1 = coupled
//	2 = starting
//	3 = running
//	4 = aborted
// 	5 = no hardware connected
//  6 = Spare
//	7 = pointer or index error
//	8 = mapping error
//	9 = parameter error
//	10 = complete
//	Any other number = ErrorID
METHOD PUBLIC M_nCerHost : UDINT
VAR_INPUT
	bEnable: BOOL;
	bDisable: BOOL;
END_VAR
//**********************************
// Reset
//**********************************
IF _bReset THEN
	IF _bError THEN
		FB_System_M_nCerHost_fbRegSetValue(bExecute:= FALSE);
		FB_System_M_nCerHost_fbNT_Reboot(START:= FALSE); 
		FB_System_M_nCerHost_iState:= 000;
	END_IF
	M_nReset(bExecute:= _bReset);
END_IF

//**********************************
// Wait for execute
//**********************************
FB_System_M_nCerHost_fbEnable_R_TRIG(CLK:= bEnable);
IF FB_System_M_nCerHost_fbEnable_R_TRIG.Q THEN
	FB_System_M_nCerHost_fbRegSetValue(bExecute:= FALSE);
	FB_System_M_nCerHost_fbNT_Reboot(START:= FALSE); 
	FB_System_M_nCerHost_iState:= 001;
END_IF
FB_System_M_nCerHost_fbDisable_R_TRIG(CLK:= bDisable);
IF FB_System_M_nCerHost_fbDisable_R_TRIG.Q THEN
	FB_System_M_nCerHost_fbRegSetValue(bExecute:= FALSE);
	FB_System_M_nCerHost_fbNT_Reboot(START:= FALSE); 
	FB_System_M_nCerHost_iState:= 010;
END_IF


//**********************************
// State maschine
//**********************************
CASE FB_System_M_nCerHost_iState OF
	
	000:	// Do nothing
	
	001:	// Enable CerHost
			M_nCerHost:= cRUNNING;
			FB_System_M_nCerHost_sValue:= 'CeRDisp.exe';
			FB_System_M_nCerHost_fbRegSetValue(
				sNetId:= '', 
				sSubKey:= 'init', 
				sValName:= 'Launch90', 
				eValType:= REG_SZ, 
				cbData:= INT_TO_UDINT(Tc2_Standard.LEN(FB_System_M_nCerHost_sValue)), 
				pData:= ADR(FB_System_M_nCerHost_sValue), 
				bExecute:= TRUE, 
				tTimeOut:= Tc2_System.DEFAULT_ADS_TIMEOUT, 
				bBusy=> , 
				bError=> , 
				nErrId=> , 
				cbWrite=> );
		
			// Error	
			IF FB_System_M_nCerHost_fbRegSetValue.bError THEN
				M_nError(nErrorID:= FB_System_M_nCerHost_fbRegSetValue.nErrId);
				M_nCerHost:= FB_System_M_nCerHost_fbRegSetValue.nErrId;
			ELSE
				// Done
				IF NOT FB_System_M_nCerHost_fbRegSetValue.bBusy THEN
					FB_System_M_nCerHost_fbRegSetValue(bExecute:= FALSE);
					FB_System_M_nCerHost_iState:= FB_System_M_nCerHost_iState +1;
				END_IF
			END_IF
	
	002:	// Enable done
			M_nCerHost:= cRUNNING;
			FB_System_M_nCerHost_iState:= 20;

	010:	// Disable CerHost
			M_nCerHost:= cRUNNING;
			FB_System_M_nCerHost_sValue:= '_CeRDisp.exe';
			FB_System_M_nCerHost_fbRegSetValue(
				sNetId:= '', 
				sSubKey:= 'init', 
				sValName:= 'Launch90', 
				eValType:= REG_SZ, 
				cbData:= INT_TO_UDINT(Tc2_Standard.LEN(FB_System_M_nCerHost_sValue)), 
				pData:= ADR(FB_System_M_nCerHost_sValue), 
				bExecute:= TRUE, 
				tTimeOut:= Tc2_System.DEFAULT_ADS_TIMEOUT, 
				bBusy=> , 
				bError=> , 
				nErrId=> , 
				cbWrite=> );
		
			// Error	
			IF FB_System_M_nCerHost_fbRegSetValue.bError THEN
				M_nError(nErrorID:= FB_System_M_nCerHost_fbRegSetValue.nErrId);
				M_nCerHost:= FB_System_M_nCerHost_fbRegSetValue.nErrId;
			ELSE
				// Done
				IF NOT FB_System_M_nCerHost_fbRegSetValue.bBusy THEN
					FB_System_M_nCerHost_fbRegSetValue(bExecute:= FALSE);
					FB_System_M_nCerHost_iState:= FB_System_M_nCerHost_iState +1;
				END_IF
			END_IF
			
	011:	// Disable done
			M_nCerHost:= cRUNNING;
			FB_System_M_nCerHost_iState:= 20;

	020:	// Reboot
			M_nCerHost:= cRUNNING;
			FB_System_M_nCerHost_fbNT_Reboot(
				NETID:= '', 
				DELAY:= 0, 
				START:= TRUE, 
				TMOUT:= Tc2_System.DEFAULT_ADS_TIMEOUT, 
				BUSY=> , 
				ERR=> , 
				ERRID=> );
	
			// Error	
			IF FB_System_M_nCerHost_fbNT_Reboot.ERR THEN
				M_nError(nErrorID:= FB_System_M_nCerHost_fbNT_Reboot.ERRID);
				M_nCerHost:= FB_System_M_nCerHost_fbNT_Reboot.ERRID;
			END_IF
		
ELSE
	FB_System_M_nCerHost_iState:= 000;
END_CASE
END_METHOD

//	The result of the method is an unsigned double integer
//	0 = idle 
//	1 = coupled
//	2 = starting
//	3 = running
//	4 = aborted
// 	5 = no hardware connected
//  6 = Spare
//	7 = pointer or index error
//	8 = mapping error
//	9 = parameter error
//	10 = complete
//	Any other number = ErrorID
METHOD PUBLIC M_nEnable : UDINT
VAR_INPUT
END_VAR
//**********************************
// Reset
//**********************************
IF _bReset THEN
	IF NOT FB_System_M_nEnable_bDone THEN
		FB_System_M_nEnable_fb_GetDeviceIdentificationEx(bExecute:= FALSE); 
		FB_System_M_nEnable_iState:= 000;
	END_IF
	M_nReset(bExecute:= _bReset);
END_IF

// Status
IF _stDeviceIdentificationEx.strHardwareCPU = 'ARM' THEN
	_bIs_ARM:= TRUE;
ELSE
	_bIs_ARM:= FALSE;
END_IF

//**********************************
// State maschine
//**********************************
CASE FB_System_M_nEnable_iState OF
	
	000:	// Init
			FB_System_M_nEnable_fb_GetDeviceIdentificationEx(bExecute:= FALSE); 
			FB_System_M_nEnable_fbADSREAD(READ:= FALSE); 
			FB_System_M_nEnable_bDone:= FALSE;
			FB_System_M_nEnable_iState:= FB_System_M_nEnable_iState +1;
		
	001:	// Get data	
			M_nEnable:= cRUNNING;
			FB_System_M_nEnable_fb_GetDeviceIdentificationEx(bExecute:= FALSE); 
			FB_System_M_nEnable_fb_GetDeviceIdentificationEx(
				bExecute:= TRUE, 
				tTimeout:= Tc2_System.DEFAULT_ADS_TIMEOUT, 
				sNetId:= '', 
				bBusy=> , 
				bError=> , 
				nErrorID=> , 
				stDevIdent=> FB_System_M_nEnable_stDeviceIdentificationEx);
	
			FB_System_M_nEnable_iState:= FB_System_M_nEnable_iState +1;
	
	002:	// Get data done
			M_nEnable:= cRUNNING;
			FB_System_M_nEnable_fb_GetDeviceIdentificationEx(bExecute:= TRUE, stDevIdent=> FB_System_M_nEnable_stDeviceIdentificationEx);
			IF FB_System_M_nEnable_fb_GetDeviceIdentificationEx.bError THEN
				M_nError(nErrorID:= FB_System_M_nEnable_fb_GetDeviceIdentificationEx.nErrorID);
				M_nEnable:= FB_System_M_nEnable_fb_GetDeviceIdentificationEx.nErrorID;
			ELSE
				// Done
				IF NOT FB_System_M_nEnable_fb_GetDeviceIdentificationEx.bBusy THEN
					_stDeviceIdentificationEx:= FB_System_M_nEnable_stDeviceIdentificationEx;
					FB_System_M_nEnable_fb_GetDeviceIdentificationEx(bExecute:= FALSE); 
					FB_System_M_nEnable_iState:= FB_System_M_nEnable_iState +1;
				END_IF	
			END_IF
		
	003:	// Read 
			FB_System_M_nEnable_fbADSREAD(
				NETID:= , 
				PORT:= 10000, 
				IDXGRP:= 160, 
				IDXOFFS:= 0, 
				LEN:= SIZEOF(FB_System_M_nEnable_arrUINT), 
				DESTADDR:= ADR(FB_System_M_nEnable_arrUINT), 
				READ:= TRUE, 
				TMOUT:= , 
				BUSY=> , 
				ERR=> , 
				ERRID=> );
						
			IF NOT FB_System_M_nEnable_fbADSREAD.BUSY THEN
				_sTwinCAT_Version:= 'v';
				_sTwinCAT_Version:= Tc2_Standard.CONCAT(_sTwinCAT_Version, UINT_TO_STRING(FB_System_M_nEnable_arrUINT[2]));
				_sTwinCAT_Version:= Tc2_Standard.CONCAT(_sTwinCAT_Version, '.');
				_sTwinCAT_Version:= Tc2_Standard.CONCAT(_sTwinCAT_Version, UINT_TO_STRING(FB_System_M_nEnable_arrUINT[1]));
				_sTwinCAT_Version:= Tc2_Standard.CONCAT(_sTwinCAT_Version, '.');
				_sTwinCAT_Version:= Tc2_Standard.CONCAT(_sTwinCAT_Version, UINT_TO_STRING(FB_System_M_nEnable_arrUINT[4]));
				_sTwinCAT_Version:= Tc2_Standard.CONCAT(_sTwinCAT_Version, '.');
				_sTwinCAT_Version:= Tc2_Standard.CONCAT(_sTwinCAT_Version, UINT_TO_STRING(FB_System_M_nEnable_arrUINT[3]));
				FB_System_M_nEnable_iState:= FB_System_M_nEnable_iState +1;
			END_IF

	004:	// Done	
			M_nEnable:= cCOMPLETE;
			FB_System_M_nEnable_bDone:= TRUE;

ELSE
	FB_System_M_nEnable_iState:= 000;
END_CASE


// bReady
IF FB_System_M_nEnable_bDone THEN
	_bReady:= TRUE;
ELSE
	_bReady:= FALSE;
END_IF
END_METHOD

METHOD PUBLIC M_nGetTimeStampInMs : ULINT
VAR_INPUT
END_VAR
M_nGetTimeStampInMs:= Tc2_EtherCAT.F_GetCurDcTaskTime64() / EC_DCTIME_TICKSPERMSEC64;
END_METHOD

PROPERTY PUBLIC P_bIs_ARM : BOOL
GET
P_bIs_ARM:= _bIs_ARM;
END_GET
END_PROPERTY

PROPERTY PUBLIC P_bIs_CE_Device : BOOL
GET
P_bIs_CE_Device:= _stDeviceIdentificationEx.strImageOsName = 'Windows CE';
END_GET
END_PROPERTY

PROPERTY PUBLIC P_bIs_x64 : BOOL
GET
IF _bIs_ARM THEN
	P_bIs_x64:= FALSE;
ELSE
	IF SIZEOF(pInternPointer) > 4 THEN
		P_bIs_x64:= TRUE;
	ELSE
		P_bIs_x64:= FALSE;
	END_IF	
END_IF
END_GET
END_PROPERTY

PROPERTY PUBLIC P_bIs_x86 : BOOL
GET
IF _bIs_ARM THEN
	P_bIs_x86:= FALSE;
ELSE
	IF SIZEOF(pInternPointer) = 4 THEN
		P_bIs_x86:= TRUE;
	ELSE
		P_bIs_x86:= FALSE;
	END_IF	
END_IF
END_GET
END_PROPERTY

PROPERTY PUBLIC P_nAdsPort : UINT
GET
P_nAdsPort:= TwinCAT_SystemInfoVarList._AppInfo.AdsPort;
END_GET
END_PROPERTY

PROPERTY PUBLIC P_nCycleTime : UDINT
GET
P_nCycleTime:= TwinCAT_SystemInfoVarList._TaskInfo[Tc2_System.GETCURTASKINDEXEX()].CycleTime;
END_GET
END_PROPERTY

PROPERTY PUBLIC P_stDeviceIdentificationEx : Tc2_Utilities.ST_DeviceIdentificationEx
GET
P_stDeviceIdentificationEx:= _stDeviceIdentificationEx;
END_GET
END_PROPERTY

PROPERTY PUBLIC P_sTwinCAT_Version : STRING
GET
P_sTwinCAT_Version:= _sTwinCAT_Version;
END_GET
END_PROPERTY

END_FUNCTION_BLOCK
